LIN {X 0,Y 573.271,Z 400.076,A -85,B 0,C 180,E1 -2125.671,E2 -2125.671} C_VEL
LIN {X 0,Y 573.245,Z 400.079,A -85,B 0,C 180,E1 -2128.184,E2 -2128.184} C_VEL
LIN {X 0,Y 573.268,Z 400.071,A -85,B 0,C 180,E1 -2130.634,E2 -2130.634} C_VEL
LIN {X 0,Y 573.241,Z 400.078,A -85,B 0,C 180,E1 -2133.508,E2 -2133.508} C_VEL
LIN {X 0,Y 573.231,Z 400.08,A -85,B 0,C 180,E1 -2136.134,E2 -2136.134} C_VEL
LIN {X 0,Y 573.255,Z 400.074,A -85,B 0,C 180,E1 -2139.174,E2 -2139.174} C_VEL
LIN {X 0,Y 573.225,Z 400.08,A -85,B 0,C 180,E1 -2141.411,E2 -2141.411} C_VEL
LIN {X 0,Y 573.248,Z 400.081,A -85,B 0,C 180,E1 -2143.621,E2 -2143.621} C_VEL
LIN {X 0,Y 573.277,Z 400.078,A -85,B 0,C 180,E1 -2145.807,E2 -2145.807} C_VEL
LIN {X 0,Y 573.27,Z 400.072,A -85,B 0,C 180,E1 -2148.744,E2 -2148.744} C_VEL
LIN {X 0,Y 573.289,Z 400.17,A -85,B 0,C 180,E1 -2149.099,E2 -2149.099} C_VEL
LIN {X 0,Y 573.723,Z 402.646,A -85,B 0,C 180,E1 -2149.194,E2 -2149.194} C_VEL
LIN {X 0,Y 573.631,Z 415.712,A -85,B 0,C 180,E1 -2149.767,E2 -2149.767} C_VEL
LIN {X 0,Y 573.485,Z 426.532,A -85,B 0,C 180,E1 -2150.388,E2 -2150.388} C_VEL
LIN {X 0,Y 573.341,Z 436.494,A -85,B 0,C 180,E1 -2151.097,E2 -2151.097} C_VEL
LIN {X 0,Y 573.294,Z 445.705,A -85,B 0,C 180,E1 -2151.895,E2 -2151.895} C_VEL
LIN {X 0,Y 573.193,Z 454.155,A -85,B 0,C 180,E1 -2152.78,E2 -2152.78} C_VEL
LIN {X 0,Y 573.148,Z 462.359,A -85,B 0,C 180,E1 -2153.841,E2 -2153.841} C_VEL
LIN {X 0,Y 573.024,Z 467.955,A -85,B 0,C 180,E1 -2154.722,E2 -2154.722} C_VEL
LIN {X 0,Y 573.036,Z 473.419,A -85,B 0,C 180,E1 -2155.78,E2 -2155.78} C_VEL
LIN {X 0,Y 573.011,Z 477.698,A -85,B 0,C 180,E1 -2156.836,E2 -2156.836} C_VEL
LIN {X 0,Y 572.952,Z 480.925,A -85,B 0,C 180,E1 -2157.891,E2 -2157.891} C_VEL
LIN {X 0,Y 572.949,Z 482.571,A -85,B 0,C 180,E1 -2158.594,E2 -2158.594} C_VEL
LIN {X 0,Y 572.941,Z 483.756,A -85,B 0,C 180,E1 -2159.297,E2 -2159.297} C_VEL
LIN {X 0,Y 572.94,Z 484.933,A -85,B 0,C 180,E1 -2160.703,E2 -2160.703} C_VEL
LIN {X 0,Y 572.946,Z 484.929,A -85,B 0,C 180,E1 -2161.406,E2 -2161.406} C_VEL
LIN {X 0,Y 572.955,Z 483.726,A -85,B 0,C 180,E1 -2162.812,E2 -2162.812} C_VEL
LIN {X 0,Y 573.009,Z 482.529,A -85,B 0,C 180,E1 -2163.516,E2 -2163.516} C_VEL
LIN {X 0,Y 573.005,Z 479.934,A -85,B 0,C 180,E1 -2164.573,E2 -2164.573} C_VEL
LIN {X 0,Y 573.051,Z 476.328,A -85,B 0,C 180,E1 -2165.63,E2 -2165.63} C_VEL
LIN {X 0,Y 573.059,Z 471.604,A -85,B 0,C 180,E1 -2166.691,E2 -2166.691} C_VEL
LIN {X 0,Y 573.087,Z 465.621,A -85,B 0,C 180,E1 -2167.753,E2 -2167.753} C_VEL
LIN {X 0,Y 573.158,Z 458.145,A -85,B 0,C 180,E1 -2168.817,E2 -2168.817} C_VEL
LIN {X 0,Y 573.217,Z 450.542,A -85,B 0,C 180,E1 -2169.705,E2 -2169.705} C_VEL
LIN {X 0,Y 573.342,Z 441.353,A -85,B 0,C 180,E1 -2170.595,E2 -2170.595} C_VEL
LIN {X 0,Y 573.451,Z 430.069,A -85,B 0,C 180,E1 -2171.469,E2 -2171.469} C_VEL
LIN {X 0,Y 573.555,Z 419.634,A -85,B 0,C 180,E1 -2172.113,E2 -2172.113} C_VEL
LIN {X 0,Y 573.669,Z 407.697,A -85,B 0,C 180,E1 -2172.694,E2 -2172.694} C_VEL
LIN {X 0,Y 573.7,Z 402.018,A -85,B 0,C 180,E1 -2172.919,E2 -2172.919} C_VEL
LIN {X 0,Y 573.284,Z 400.077,A -85,B 0,C 180,E1 -2172.996,E2 -2172.996} C_VEL
LIN {X 0,Y 573.244,Z 400.08,A -85,B 0,C 180,E1 -2175.648,E2 -2175.648} C_VEL
LIN {X 0,Y 573.243,Z 400.081,A -85,B 0,C 180,E1 -2177.849,E2 -2177.849} C_VEL
LIN {X 0,Y 573.256,Z 400.082,A -85,B 0,C 180,E1 -2180.076,E2 -2180.076} C_VEL
LIN {X 0,Y 573.239,Z 400.084,A -85,B 0,C 180,E1 -2183.099,E2 -2183.099} C_VEL
LIN {X 0,Y 573.26,Z 400.078,A -85,B 0,C 180,E1 -2185.41,E2 -2185.41} C_VEL
LIN {X 0,Y 573.257,Z 400.077,A -85,B 0,C 180,E1 -2188.029,E2 -2188.029} C_VEL
LIN {X 0,Y 573.251,Z 400.081,A -85,B 0,C 180,E1 -2190.176,E2 -2190.176} C_VEL
LIN {X 0,Y 573.258,Z 400.081,A -85,B 0,C 180,E1 -2192.645,E2 -2192.645} C_VEL
LIN {X 0,Y 573.211,Z 400.084,A -85,B 0,C 180,E1 -2195.188,E2 -2195.188} C_VEL
LIN {X 0,Y 573.238,Z 400.08,A -85,B 0,C 180,E1 -2197.807,E2 -2197.807} C_VEL
LIN {X 0,Y 573.248,Z 400.079,A -85,B 0,C 180,E1 -2200.525,E2 -2200.525} C_VEL
LIN {X 0,Y 573.252,Z 400.078,A -85,B 0,C 180,E1 -2203.358,E2 -2203.358} C_VEL
LIN {X 0,Y 573.243,Z 400.08,A -85,B 0,C 180,E1 -2206.331,E2 -2206.331} C_VEL
LIN {X 0,Y 573.274,Z 400.079,A -85,B 0,C 180,E1 -2209.472,E2 -2209.472} C_VEL
LIN {X 0,Y 573.24,Z 400.084,A -85,B 0,C 180,E1 -2212.192,E2 -2212.192} C_VEL
LIN {X 0,Y 573.309,Z 400.2,A -85,B 0,C 180,E1 -2213.383,E2 -2213.383} C_VEL
LIN {X 0,Y 573.995,Z 405.053,A -85,B 0,C 180,E1 -2214.437,E2 -2214.437} C_VEL
LIN {X 0,Y 573.917,Z 418.715,A -85,B 0,C 180,E1 -2217.189,E2 -2217.189} C_VEL
LIN {X 0,Y 573.925,Z 434.068,A -85,B 0,C 180,E1 -2220.168,E2 -2220.168} C_VEL
LIN {X 0,Y 573.92,Z 449.451,A -85,B 0,C 180,E1 -2223.058,E2 -2223.058} C_VEL
LIN {X 0,Y 573.821,Z 461.449,A -85,B 0,C 180,E1 -2225.391,E2 -2225.391} C_VEL
LIN {X 0,Y 573.637,Z 475.144,A -85,B 0,C 180,E1 -2228.057,E2 -2228.057} C_VEL
LIN {X 0,Y 573.502,Z 488.839,A -85,B 0,C 180,E1 -2230.678,E2 -2230.678} C_VEL
LIN {X 0,Y 573.363,Z 502.686,A -85,B 0,C 180,E1 -2233.287,E2 -2233.287} C_VEL
LIN {X 0,Y 573.252,Z 518.186,A -85,B 0,C 180,E1 -2236.168,E2 -2236.168} C_VEL
LIN {X 0,Y 573.191,Z 525.155,A -85,B 0,C 180,E1 -2237.452,E2 -2237.452} C_VEL
LIN {X 0,Y 573.863,Z 530.936,A -85,B 0,C 180,E1 -2237.557,E2 -2237.557} C_VEL
LIN {X 0,Y 573.81,Z 544.212,A -85,B 0,C 180,E1 -2237.87,E2 -2237.87} C_VEL
LIN {X 0,Y 573.714,Z 556.368,A -85,B 0,C 180,E1 -2238.294,E2 -2238.294} C_VEL
LIN {X 0,Y 573.586,Z 568.658,A -85,B 0,C 180,E1 -2238.875,E2 -2238.875} C_VEL
LIN {X 0,Y 573.434,Z 580.2,A -85,B 0,C 180,E1 -2239.585,E2 -2239.585} C_VEL
LIN {X 0,Y 573.334,Z 590.597,A -85,B 0,C 180,E1 -2240.385,E2 -2240.385} C_VEL
LIN {X 0,Y 573.241,Z 599.11,A -85,B 0,C 180,E1 -2241.184,E2 -2241.184} C_VEL
LIN {X 0,Y 573.161,Z 606.959,A -85,B 0,C 180,E1 -2242.071,E2 -2242.071} C_VEL
LIN {X 0,Y 573.073,Z 614.953,A -85,B 0,C 180,E1 -2243.185,E2 -2243.185} C_VEL
LIN {X 0,Y 573.07,Z 621.679,A -85,B 0,C 180,E1 -2244.369,E2 -2244.369} C_VEL
LIN {X 0,Y 573.029,Z 626.371,A -85,B 0,C 180,E1 -2245.427,E2 -2245.427} C_VEL
LIN {X 0,Y 573.022,Z 629.956,A -85,B 0,C 180,E1 -2246.484,E2 -2246.484} C_VEL
LIN {X 0,Y 572.959,Z 631.808,A -85,B 0,C 180,E1 -2247.188,E2 -2247.188} C_VEL
LIN {X 0,Y 572.938,Z 633.199,A -85,B 0,C 180,E1 -2247.891,E2 -2247.891} C_VEL
LIN {X 0,Y 572.941,Z 634.785,A -85,B 0,C 180,E1 -2249.297,E2 -2249.297} C_VEL
LIN {X 0,Y 572.938,Z 635,A -85,B 0,C 180,E1 -2250,E2 -2250} C_VEL
LIN {X 0,Y 572.946,Z 634.186,A -85,B 0,C 180,E1 -2251.406,E2 -2251.406} C_VEL
LIN {X 0,Y 572.938,Z 633.2,A -85,B 0,C 180,E1 -2252.109,E2 -2252.109} C_VEL
LIN {X 0,Y 572.959,Z 631.81,A -85,B 0,C 180,E1 -2252.812,E2 -2252.812} C_VEL
LIN {X 0,Y 573.014,Z 628.896,A -85,B 0,C 180,E1 -2253.868,E2 -2253.868} C_VEL
LIN {X 0,Y 572.963,Z 624.95,A -85,B 0,C 180,E1 -2254.925,E2 -2254.925} C_VEL
LIN {X 0,Y 573.064,Z 618.878,A -85,B 0,C 180,E1 -2256.16,E2 -2256.16} C_VEL
LIN {X 0,Y 573.119,Z 612.238,A -85,B 0,C 180,E1 -2257.221,E2 -2257.221} C_VEL
LIN {X 0,Y 573.201,Z 603.991,A -85,B 0,C 180,E1 -2258.283,E2 -2258.283} C_VEL
LIN {X 0,Y 573.287,Z 595.539,A -85,B 0,C 180,E1 -2259.17,E2 -2259.17} C_VEL
LIN {X 0,Y 573.42,Z 585.098,A -85,B 0,C 180,E1 -2260.058,E2 -2260.058} C_VEL
LIN {X 0,Y 573.555,Z 573.44,A -85,B 0,C 180,E1 -2260.852,E2 -2260.852} C_VEL
LIN {X 0,Y 573.65,Z 562.318,A -85,B 0,C 180,E1 -2261.446,E2 -2261.446} C_VEL
LIN {X 0,Y 573.731,Z 549.177,A -85,B 0,C 180,E1 -2261.974,E2 -2261.974} C_VEL
LIN {X 0,Y 573.854,Z 536.524,A -85,B 0,C 180,E1 -2262.331,E2 -2262.331} C_VEL
LIN {X 0,Y 573.611,Z 527.738,A -85,B 0,C 180,E1 -2262.499,E2 -2262.499} C_VEL
LIN {X 0,Y 573.194,Z 525.035,A -85,B 0,C 180,E1 -2262.57,E2 -2262.57} C_VEL
LIN {X 0,Y 573.316,Z 510.362,A -85,B 0,C 180,E1 -2265.281,E2 -2265.281} C_VEL
LIN {X 0,Y 573.46,Z 494.71,A -85,B 0,C 180,E1 -2268.211,E2 -2268.211} C_VEL
LIN {X 0,Y 573.597,Z 479.542,A -85,B 0,C 180,E1 -2271.096,E2 -2271.096} C_VEL
LIN {X 0,Y 573.775,Z 465.364,A -85,B 0,C 180,E1 -2273.841,E2 -2273.841} C_VEL
LIN {X 0,Y 573.939,Z 451.13,A -85,B 0,C 180,E1 -2276.632,E2 -2276.632} C_VEL
LIN {X 0,Y 573.94,Z 435.25,A -85,B 0,C 180,E1 -2279.61,E2 -2279.61} C_VEL
LIN {X 0,Y 573.92,Z 421.222,A -85,B 0,C 180,E1 -2282.333,E2 -2282.333} C_VEL
LIN {X 0,Y 574.045,Z 405.153,A -85,B 0,C 180,E1 -2285.559,E2 -2285.559} C_VEL
LIN {X 0,Y 573.294,Z 400.077,A -85,B 0,C 180,E1 -2286.7,E2 -2286.7} C_VEL
LIN {X 0,Y 573.251,Z 400.081,A -85,B 0,C 180,E1 -2289.607,E2 -2289.607} C_VEL
LIN {X 0,Y 573.242,Z 400.084,A -85,B 0,C 180,E1 -2292.641,E2 -2292.641} C_VEL
LIN {X 0,Y 573.242,Z 400.084,A -85,B 0,C 180,E1 -2295.667,E2 -2295.667} C_VEL
LIN {X 0,Y 573.247,Z 400.081,A -85,B 0,C 180,E1 -2298.544,E2 -2298.544} C_VEL
LIN {X 0,Y 573.252,Z 400.082,A -85,B 0,C 180,E1 -2301.299,E2 -2301.299} C_VEL
LIN {X 0,Y 573.244,Z 400.081,A -85,B 0,C 180,E1 -2304.014,E2 -2304.014} C_VEL
LIN {X 0,Y 573.271,Z 400.08,A -85,B 0,C 180,E1 -2306.518,E2 -2306.518} C_VEL
LIN {X 0,Y 573.231,Z 400.082,A -85,B 0,C 180,E1 -2309.118,E2 -2309.118} C_VEL
LIN {X 0,Y 573.266,Z 400.08,A -85,B 0,C 180,E1 -2311.969,E2 -2311.969} C_VEL
LIN {X 0,Y 573.26,Z 400.079,A -85,B 0,C 180,E1 -2314.59,E2 -2314.59} C_VEL
LIN {X 0,Y 573.24,Z 400.083,A -85,B 0,C 180,E1 -2317.662,E2 -2317.662} C_VEL
LIN {X 0,Y 573.281,Z 400.078,A -85,B 0,C 180,E1 -2320.728,E2 -2320.728} C_VEL
LIN {X 0,Y 573.257,Z 400.079,A -85,B 0,C 180,E1 -2323.622,E2 -2323.622} C_VEL
LIN {X 0,Y 573.277,Z 400.077,A -85,B 0,C 180,E1 -2325.807,E2 -2325.807} C_VEL
LIN {X 0,Y 573.265,Z 400.078,A -85,B 0,C 180,E1 -2328.745,E2 -2328.745} C_VEL
LIN {X 0,Y 573.257,Z 400.081,A -85,B 0,C 180,E1 -2331.54,E2 -2331.54} C_VEL
LIN {X 0,Y 573.248,Z 400.082,A -85,B 0,C 180,E1 -2333.665,E2 -2333.665} C_VEL
LIN {X 0,Y 573.234,Z 400.084,A -85,B 0,C 180,E1 -2335.782,E2 -2335.782} C_VEL
LIN {X 0,Y 573.317,Z 400.073,A -85,B 0,C 180,E1 -2337.893,E2 -2337.893} C_VEL
LIN {X 0,Y 573.337,Z 400.069,A -85,B 0,C 180,E1 -2340.702,E2 -2340.702} C_VEL
LIN {X 0,Y 573.235,Z 400.085,A -85,B 0,C 180,E1 -2343.515,E2 -2343.515} C_VEL
LIN {X 0,Y 573.291,Z 400.078,A -85,B 0,C 180,E1 -2345.628,E2 -2345.628} C_VEL
LIN {X 0,Y 573.294,Z 400.075,A -85,B 0,C 180,E1 -2348.46,E2 -2348.46} C_VEL
LIN {X 0,Y 573.275,Z 400.078,A -85,B 0,C 180,E1 -2351.312,E2 -2351.312} C_VEL
LIN {X 0,Y 573.277,Z 400.079,A -85,B 0,C 180,E1 -2354.193,E2 -2354.193} C_VEL
LIN {X 0,Y 573.261,Z 400.078,A -85,B 0,C 180,E1 -2357.112,E2 -2357.112} C_VEL
LIN {X 0,Y 573.259,Z 400.079,A -85,B 0,C 180,E1 -2360.077,E2 -2360.077} C_VEL
LIN {X 0,Y 573.242,Z 400.081,A -85,B 0,C 180,E1 -2362.338,E2 -2362.338} C_VEL
LIN {X 0,Y 573.254,Z 400.078,A -85,B 0,C 180,E1 -2364.393,E2 -2364.393} C_VEL
LIN {X 0,Y 572.627,Z 400.159,A -85,B 0,C 180,E1 -2364.98,E2 -2364.98} C_VEL
LIN {X 0,Y 569.784,Z 400.516,A -85,B 0,C 180,E1 -2365.931,E2 -2365.931} C_VEL
LIN {X 0,Y 567.351,Z 400.819,A -85,B 0,C 180,E1 -2366.697,E2 -2366.697} C_VEL
LIN {X 0,Y 566.296,Z 400.949,A -85,B 0,C 180,E1 -2367.288,E2 -2367.288} C_VEL
LIN {X 0,Y 566.206,Z 400.959,A -85,B 0,C 180,E1 -2367.488,E2 -2367.488} C_VEL
LIN {X 0,Y 566.204,Z 400.959,A -85,B 0,C 180,E1 -2369.769,E2 -2369.769} C_VEL
LIN {X 0,Y 566.209,Z 400.958,A -85,B 0,C 180,E1 -2372.431,E2 -2372.431} C_VEL
LIN {X 0,Y 566.206,Z 400.959,A -85,B 0,C 180,E1 -2374.993,E2 -2374.993} C_VEL
LIN {X 0,Y 566.2,Z 400.958,A -85,B 0,C 180,E1 -2377.461,E2 -2377.461} C_VEL
LIN {X 0,Y 566.21,Z 400.959,A -85,B 0,C 180,E1 -2380.199,E2 -2380.199} C_VEL
LIN {X 0,Y 566.209,Z 400.957,A -85,B 0,C 180,E1 -2383.054,E2 -2383.054} C_VEL
LIN {X 0,Y 566.206,Z 400.958,A -85,B 0,C 180,E1 -2386.048,E2 -2386.048} C_VEL
LIN {X 0,Y 566.215,Z 400.958,A -85,B 0,C 180,E1 -2388.864,E2 -2388.864} C_VEL
LIN {X 0,Y 566.193,Z 400.959,A -85,B 0,C 180,E1 -2391.637,E2 -2391.637} C_VEL
LIN {X 0,Y 566.204,Z 400.96,A -85,B 0,C 180,E1 -2394.311,E2 -2394.311} C_VEL
LIN {X 0,Y 566.234,Z 400.954,A -85,B 0,C 180,E1 -2396.899,E2 -2396.899} C_VEL
LIN {X 0,Y 566.199,Z 400.959,A -85,B 0,C 180,E1 -2399.408,E2 -2399.408} C_VEL
LIN {X 0,Y 566.216,Z 400.959,A -85,B 0,C 180,E1 -2401.858,E2 -2401.858} C_VEL
LIN {X 0,Y 566.217,Z 400.957,A -85,B 0,C 180,E1 -2404.251,E2 -2404.251} C_VEL
LIN {X 0,Y 566.178,Z 400.96,A -85,B 0,C 180,E1 -2406.718,E2 -2406.718} C_VEL
LIN {X 0,Y 566.219,Z 400.958,A -85,B 0,C 180,E1 -2409.663,E2 -2409.663} C_VEL
LIN {X 0,Y 566.208,Z 400.959,A -85,B 0,C 180,E1 -2412.669,E2 -2412.669} C_VEL
LIN {X 0,Y 566.239,Z 400.954,A -85,B 0,C 180,E1 -2415.627,E2 -2415.627} C_VEL
LIN {X 0,Y 566.24,Z 400.953,A -85,B 0,C 180,E1 -2418.675,E2 -2418.675} C_VEL
LIN {X 0,Y 566.232,Z 400.955,A -85,B 0,C 180,E1 -2420.962,E2 -2420.962} C_VEL
LIN {X 0,Y 566.753,Z 404.787,A -85,B 0,C 180,E1 -2421.128,E2 -2421.128} C_VEL
LIN {X 0,Y 566.621,Z 417.32,A -85,B 0,C 180,E1 -2421.71,E2 -2421.71} C_VEL
LIN {X 0,Y 566.484,Z 427.742,A -85,B 0,C 180,E1 -2422.336,E2 -2422.336} C_VEL
LIN {X 0,Y 566.34,Z 436.703,A -85,B 0,C 180,E1 -2422.99,E2 -2422.99} C_VEL
LIN {X 0,Y 566.196,Z 445.6,A -85,B 0,C 180,E1 -2423.765,E2 -2423.765} C_VEL
LIN {X 0,Y 566.157,Z 455.476,A -85,B 0,C 180,E1 -2424.837,E2 -2424.837} C_VEL
LIN {X 0,Y 566.084,Z 463.43,A -85,B 0,C 180,E1 -2425.906,E2 -2425.906} C_VEL
LIN {X 0,Y 566.013,Z 468.831,A -85,B 0,C 180,E1 -2426.797,E2 -2426.797} C_VEL
LIN {X 0,Y 565.885,Z 474.122,A -85,B 0,C 180,E1 -2427.865,E2 -2427.865} C_VEL
LIN {X 0,Y 565.912,Z 478.247,A -85,B 0,C 180,E1 -2428.933,E2 -2428.933} C_VEL
LIN {X 0,Y 565.844,Z 481.333,A -85,B 0,C 180,E1 -2430,E2 -2430} C_VEL
LIN {X 0,Y 565.841,Z 482.847,A -85,B 0,C 180,E1 -2430.712,E2 -2430.712} C_VEL
LIN {X 0,Y 565.839,Z 484.657,A -85,B 0,C 180,E1 -2432.136,E2 -2432.136} C_VEL
LIN {X 0,Y 565.911,Z 484.894,A -85,B 0,C 180,E1 -2433.56,E2 -2433.56} C_VEL
LIN {X 0,Y 565.912,Z 484.393,A -85,B 0,C 180,E1 -2434.273,E2 -2434.273} C_VEL
LIN {X 0,Y 565.851,Z 483.503,A -85,B 0,C 180,E1 -2434.988,E2 -2434.988} C_VEL
LIN {X 0,Y 565.899,Z 480.492,A -85,B 0,C 180,E1 -2436.418,E2 -2436.418} C_VEL
LIN {X 0,Y 565.922,Z 477.065,A -85,B 0,C 180,E1 -2437.493,E2 -2437.493} C_VEL
LIN {X 0,Y 565.954,Z 472.52,A -85,B 0,C 180,E1 -2438.57,E2 -2438.57} C_VEL
LIN {X 0,Y 566.005,Z 466.736,A -85,B 0,C 180,E1 -2439.65,E2 -2439.65} C_VEL
LIN {X 0,Y 566.064,Z 459.561,A -85,B 0,C 180,E1 -2440.733,E2 -2440.733} C_VEL
LIN {X 0,Y 566.191,Z 450.536,A -85,B 0,C 180,E1 -2441.819,E2 -2441.819} C_VEL
LIN {X 0,Y 566.295,Z 441.228,A -85,B 0,C 180,E1 -2442.726,E2 -2442.726} C_VEL
LIN {X 0,Y 566.42,Z 430.825,A -85,B 0,C 180,E1 -2443.544,E2 -2443.544} C_VEL
LIN {X 0,Y 566.56,Z 420.83,A -85,B 0,C 180,E1 -2444.182,E2 -2444.182} C_VEL
LIN {X 0,Y 566.719,Z 409.031,A -85,B 0,C 180,E1 -2444.784,E2 -2444.784} C_VEL
LIN {X 0,Y 566.786,Z 403.376,A -85,B 0,C 180,E1 -2445.016,E2 -2445.016} C_VEL
LIN {X 0,Y 566.244,Z 400.951,A -85,B 0,C 180,E1 -2445.131,E2 -2445.131} C_VEL
LIN {X 0,Y 566.2,Z 400.957,A -85,B 0,C 180,E1 -2448.078,E2 -2448.078} C_VEL
LIN {X 0,Y 566.213,Z 400.959,A -85,B 0,C 180,E1 -2450.337,E2 -2450.337} C_VEL
LIN {X 0,Y 566.175,Z 400.954,A -85,B 0,C 180,E1 -2453.281,E2 -2453.281} C_VEL
LIN {X 0,Y 566.219,Z 400.951,A -85,B 0,C 180,E1 -2455.749,E2 -2455.749} C_VEL
LIN {X 0,Y 566.208,Z 400.959,A -85,B 0,C 180,E1 -2458.202,E2 -2458.202} C_VEL
LIN {X 0,Y 566.196,Z 400.952,A -85,B 0,C 180,E1 -2461.076,E2 -2461.076} C_VEL
LIN {X 0,Y 566.218,Z 400.951,A -85,B 0,C 180,E1 -2463.734,E2 -2463.734} C_VEL
LIN {X 0,Y 566.213,Z 400.953,A -85,B 0,C 180,E1 -2466.569,E2 -2466.569} C_VEL
LIN {X 0,Y 566.221,Z 400.951,A -85,B 0,C 180,E1 -2469.686,E2 -2469.686} C_VEL
LIN {X 0,Y 566.206,Z 400.95,A -85,B 0,C 180,E1 -2472.917,E2 -2472.917} C_VEL
LIN {X 0,Y 566.208,Z 400.96,A -85,B 0,C 180,E1 -2476.048,E2 -2476.048} C_VEL
LIN {X 0,Y 566.187,Z 400.953,A -85,B 0,C 180,E1 -2478.861,E2 -2478.861} C_VEL
LIN {X 0,Y 566.19,Z 400.956,A -85,B 0,C 180,E1 -2481.637,E2 -2481.637} C_VEL
LIN {X 0,Y 566.167,Z 400.959,A -85,B 0,C 180,E1 -2484.308,E2 -2484.308} C_VEL
LIN {X 0,Y 566.225,Z 400.948,A -85,B 0,C 180,E1 -2486.898,E2 -2486.898} C_VEL
LIN {X 0,Y 566.185,Z 400.955,A -85,B 0,C 180,E1 -2489.407,E2 -2489.407} C_VEL
LIN {X 0,Y 566.217,Z 400.959,A -85,B 0,C 180,E1 -2491.857,E2 -2491.857} C_VEL
LIN {X 0,Y 566.218,Z 400.952,A -85,B 0,C 180,E1 -2494.251,E2 -2494.251} C_VEL
LIN {X 0,Y 566.173,Z 400.954,A -85,B 0,C 180,E1 -2496.719,E2 -2496.719} C_VEL
LIN {X 0,Y 566.212,Z 400.958,A -85,B 0,C 180,E1 -2499.663,E2 -2499.663} C_VEL
LIN {X 0,Y 566.204,Z 400.95,A -85,B 0,C 180,E1 -2502.668,E2 -2502.668} C_VEL
LIN {X 0,Y 566.239,Z 400.955,A -85,B 0,C 180,E1 -2505.627,E2 -2505.627} C_VEL
LIN {X 0,Y 566.242,Z 400.948,A -85,B 0,C 180,E1 -2508.674,E2 -2508.674} C_VEL
LIN {X 0,Y 566.239,Z 401.02,A -85,B 0,C 180,E1 -2508.978,E2 -2508.978} C_VEL
LIN {X 0,Y 566.766,Z 403.757,A -85,B 0,C 180,E1 -2509.087,E2 -2509.087} C_VEL
LIN {X 0,Y 566.661,Z 415.97,A -85,B 0,C 180,E1 -2509.64,E2 -2509.64} C_VEL
LIN {X 0,Y 566.506,Z 426.717,A -85,B 0,C 180,E1 -2510.268,E2 -2510.268} C_VEL
LIN {X 0,Y 566.338,Z 436.65,A -85,B 0,C 180,E1 -2510.986,E2 -2510.986} C_VEL
LIN {X 0,Y 566.262,Z 445.838,A -85,B 0,C 180,E1 -2511.794,E2 -2511.794} C_VEL
LIN {X 0,Y 566.119,Z 455.757,A -85,B 0,C 180,E1 -2512.869,E2 -2512.869} C_VEL
LIN {X 0,Y 566.084,Z 463.615,A -85,B 0,C 180,E1 -2513.942,E2 -2513.942} C_VEL
LIN {X 0,Y 565.915,Z 469.96,A -85,B 0,C 180,E1 -2515.013,E2 -2515.013} C_VEL
LIN {X 0,Y 565.947,Z 475.023,A -85,B 0,C 180,E1 -2516.084,E2 -2516.084} C_VEL
LIN {X 0,Y 565.914,Z 480.041,A -85,B 0,C 180,E1 -2517.509,E2 -2517.509} C_VEL
LIN {X 0,Y 565.849,Z 482.599,A -85,B 0,C 180,E1 -2518.576,E2 -2518.576} C_VEL
LIN {X 0,Y 565.841,Z 483.775,A -85,B 0,C 180,E1 -2519.288,E2 -2519.288} C_VEL
LIN {X 0,Y 565.84,Z 484.936,A -85,B 0,C 180,E1 -2520.712,E2 -2520.712} C_VEL
LIN {X 0,Y 565.846,Z 484.927,A -85,B 0,C 180,E1 -2521.423,E2 -2521.423} C_VEL
LIN {X 0,Y 565.874,Z 483.704,A -85,B 0,C 180,E1 -2522.847,E2 -2522.847} C_VEL
LIN {X 0,Y 565.915,Z 482.505,A -85,B 0,C 180,E1 -2523.56,E2 -2523.56} C_VEL
LIN {X 0,Y 565.896,Z 479.897,A -85,B 0,C 180,E1 -2524.63,E2 -2524.63} C_VEL
LIN {X 0,Y 565.978,Z 476.278,A -85,B 0,C 180,E1 -2525.701,E2 -2525.701} C_VEL
LIN {X 0,Y 565.973,Z 470.712,A -85,B 0,C 180,E1 -2526.936,E2 -2526.936} C_VEL
LIN {X 0,Y 566.022,Z 464.381,A -85,B 0,C 180,E1 -2528.03,E2 -2528.03} C_VEL
LIN {X 0,Y 566.108,Z 458.035,A -85,B 0,C 180,E1 -2528.927,E2 -2528.927} C_VEL
LIN {X 0,Y 566.189,Z 450.414,A -85,B 0,C 180,E1 -2529.827,E2 -2529.827} C_VEL
LIN {X 0,Y 566.324,Z 441.203,A -85,B 0,C 180,E1 -2530.728,E2 -2530.728} C_VEL
LIN {X 0,Y 566.46,Z 429.586,A -85,B 0,C 180,E1 -2531.631,E2 -2531.631} C_VEL
LIN {X 0,Y 566.571,Z 419.374,A -85,B 0,C 180,E1 -2532.265,E2 -2532.265} C_VEL
LIN {X 0,Y 566.703,Z 408.396,A -85,B 0,C 180,E1 -2532.808,E2 -2532.808} C_VEL
LIN {X 0,Y 566.671,Z 402.914,A -85,B 0,C 180,E1 -2533.036,E2 -2533.036} C_VEL
LIN {X 0,Y 566.221,Z 400.958,A -85,B 0,C 180,E1 -2533.138,E2 -2533.138} C_VEL
LIN {X 0,Y 566.21,Z 400.958,A -85,B 0,C 180,E1 -2535.847,E2 -2535.847} C_VEL
LIN {X 0,Y 566.197,Z 400.958,A -85,B 0,C 180,E1 -2538.078,E2 -2538.078} C_VEL
LIN {X 0,Y 566.218,Z 400.959,A -85,B 0,C 180,E1 -2540.337,E2 -2540.337} C_VEL
LIN {X 0,Y 566.173,Z 400.962,A -85,B 0,C 180,E1 -2543.281,E2 -2543.281} C_VEL
LIN {X 0,Y 566.22,Z 400.958,A -85,B 0,C 180,E1 -2545.749,E2 -2545.749} C_VEL
LIN {X 0,Y 566.207,Z 400.956,A -85,B 0,C 180,E1 -2548.202,E2 -2548.202} C_VEL
LIN {X 0,Y 566.195,Z 400.959,A -85,B 0,C 180,E1 -2551.076,E2 -2551.076} C_VEL
LIN {X 0,Y 566.216,Z 400.955,A -85,B 0,C 180,E1 -2553.734,E2 -2553.734} C_VEL
LIN {X 0,Y 566.204,Z 400.957,A -85,B 0,C 180,E1 -2556.57,E2 -2556.57} C_VEL
LIN {X 0,Y 566.219,Z 400.958,A -85,B 0,C 180,E1 -2559.686,E2 -2559.686} C_VEL
LIN {X 0,Y 566.21,Z 400.956,A -85,B 0,C 180,E1 -2562.918,E2 -2562.918} C_VEL
LIN {X 0,Y 566.198,Z 400.956,A -85,B 0,C 180,E1 -2566.049,E2 -2566.049} C_VEL
LIN {X 0,Y 566.224,Z 400.956,A -85,B 0,C 180,E1 -2569.212,E2 -2569.212} C_VEL
LIN {X 0,Y 566.193,Z 400.959,A -85,B 0,C 180,E1 -2571.637,E2 -2571.637} C_VEL
LIN {X 0,Y 566.245,Z 401.004,A -85,B 0,C 180,E1 -2573.156,E2 -2573.156} C_VEL
LIN {X 0,Y 567.071,Z 406.484,A -85,B 0,C 180,E1 -2574.373,E2 -2574.373} C_VEL
LIN {X 0,Y 566.969,Z 419.054,A -85,B 0,C 180,E1 -2576.947,E2 -2576.947} C_VEL
LIN {X 0,Y 566.974,Z 433.91,A -85,B 0,C 180,E1 -2579.866,E2 -2579.866} C_VEL
LIN {X 0,Y 566.924,Z 448.675,A -85,B 0,C 180,E1 -2582.698,E2 -2582.698} C_VEL
LIN {X 0,Y 566.852,Z 463.406,A -85,B 0,C 180,E1 -2585.459,E2 -2585.459} C_VEL
LIN {X 0,Y 566.653,Z 477.101,A -85,B 0,C 180,E1 -2588.156,E2 -2588.156} C_VEL
LIN {X 0,Y 566.494,Z 491.063,A -85,B 0,C 180,E1 -2590.858,E2 -2590.858} C_VEL
LIN {X 0,Y 566.335,Z 504.491,A -85,B 0,C 180,E1 -2593.416,E2 -2593.416} C_VEL
LIN {X 0,Y 566.198,Z 520.142,A -85,B 0,C 180,E1 -2596.359,E2 -2596.359} C_VEL
LIN {X 0,Y 566.153,Z 525.11,A -85,B 0,C 180,E1 -2597.285,E2 -2597.285} C_VEL
LIN {X 0,Y 566.954,Z 532.077,A -85,B 0,C 180,E1 -2597.425,E2 -2597.425} C_VEL
LIN {X 0,Y 566.831,Z 545.732,A -85,B 0,C 180,E1 -2597.764,E2 -2597.764} C_VEL
LIN {X 0,Y 566.706,Z 558.519,A -85,B 0,C 180,E1 -2598.238,E2 -2598.238} C_VEL
LIN {X 0,Y 566.561,Z 570.723,A -85,B 0,C 180,E1 -2598.853,E2 -2598.853} C_VEL
LIN {X 0,Y 566.419,Z 581.479,A -85,B 0,C 180,E1 -2599.545,E2 -2599.545} C_VEL
LIN {X 0,Y 566.301,Z 591.645,A -85,B 0,C 180,E1 -2600.355,E2 -2600.355} C_VEL
LIN {X 0,Y 566.166,Z 600.785,A -85,B 0,C 180,E1 -2601.253,E2 -2601.253} C_VEL
LIN {X 0,Y 566.081,Z 609.688,A -85,B 0,C 180,E1 -2602.33,E2 -2602.33} C_VEL
LIN {X 0,Y 565.968,Z 616.955,A -85,B 0,C 180,E1 -2603.422,E2 -2603.422} C_VEL
LIN {X 0,Y 566.004,Z 621.679,A -85,B 0,C 180,E1 -2604.299,E2 -2604.299} C_VEL
LIN {X 0,Y 565.933,Z 626.371,A -85,B 0,C 180,E1 -2605.37,E2 -2605.37} C_VEL
LIN {X 0,Y 565.927,Z 629.957,A -85,B 0,C 180,E1 -2606.44,E2 -2606.44} C_VEL
LIN {X 0,Y 565.878,Z 631.808,A -85,B 0,C 180,E1 -2607.152,E2 -2607.152} C_VEL
LIN {X 0,Y 565.846,Z 634.185,A -85,B 0,C 180,E1 -2608.576,E2 -2608.576} C_VEL
LIN {X 0,Y 565.839,Z 635,A -85,B 0,C 180,E1 -2610,E2 -2610} C_VEL
LIN {X 0,Y 565.846,Z 634.186,A -85,B 0,C 180,E1 -2611.423,E2 -2611.423} C_VEL
LIN {X 0,Y 565.878,Z 631.81,A -85,B 0,C 180,E1 -2612.847,E2 -2612.847} C_VEL
LIN {X 0,Y 565.926,Z 628.896,A -85,B 0,C 180,E1 -2613.916,E2 -2613.916} C_VEL
LIN {X 0,Y 565.878,Z 624.95,A -85,B 0,C 180,E1 -2614.987,E2 -2614.987} C_VEL
LIN {X 0,Y 566.002,Z 619.867,A -85,B 0,C 180,E1 -2616.058,E2 -2616.058} C_VEL
LIN {X 0,Y 566.04,Z 613.469,A -85,B 0,C 180,E1 -2617.132,E2 -2617.132} C_VEL
LIN {X 0,Y 566.133,Z 605.479,A -85,B 0,C 180,E1 -2618.208,E2 -2618.208} C_VEL
LIN {X 0,Y 566.229,Z 597.337,A -85,B 0,C 180,E1 -2619.105,E2 -2619.105} C_VEL
LIN {X 0,Y 566.342,Z 587.402,A -85,B 0,C 180,E1 -2620.005,E2 -2620.005} C_VEL
LIN {X 0,Y 566.528,Z 576.292,A -85,B 0,C 180,E1 -2620.807,E2 -2620.807} C_VEL
LIN {X 0,Y 566.612,Z 565.179,A -85,B 0,C 180,E1 -2621.447,E2 -2621.447} C_VEL
LIN {X 0,Y 566.73,Z 552.987,A -85,B 0,C 180,E1 -2621.988,E2 -2621.988} C_VEL
LIN {X 0,Y 566.887,Z 540.181,A -85,B 0,C 180,E1 -2622.394,E2 -2622.394} C_VEL
LIN {X 0,Y 566.761,Z 528.952,A -85,B 0,C 180,E1 -2622.634,E2 -2622.634} C_VEL
LIN {X 0,Y 566.155,Z 525.035,A -85,B 0,C 180,E1 -2622.729,E2 -2622.729} C_VEL
LIN {X 0,Y 566.283,Z 510.362,A -85,B 0,C 180,E1 -2625.476,E2 -2625.476} C_VEL
LIN {X 0,Y 566.459,Z 494.71,A -85,B 0,C 180,E1 -2628.444,E2 -2628.444} C_VEL
LIN {X 0,Y 566.61,Z 479.879,A -85,B 0,C 180,E1 -2631.303,E2 -2631.303} C_VEL
LIN {X 0,Y 566.812,Z 467.322,A -85,B 0,C 180,E1 -2633.764,E2 -2633.764} C_VEL
LIN {X 0,Y 566.898,Z 457.181,A -85,B 0,C 180,E1 -2635.716,E2 -2635.716} C_VEL
LIN {X 0,Y 566.935,Z 441.919,A -85,B 0,C 180,E1 -2638.584,E2 -2638.584} C_VEL
LIN {X 0,Y 566.972,Z 427.582,A -85,B 0,C 180,E1 -2641.374,E2 -2641.374} C_VEL
LIN {X 0,Y 567.049,Z 411.805,A -85,B 0,C 180,E1 -2644.543,E2 -2644.543} C_VEL
LIN {X 0,Y 567.006,Z 405.049,A -85,B 0,C 180,E1 -2645.949,E2 -2645.949} C_VEL
LIN {X 0,Y 566.226,Z 400.958,A -85,B 0,C 180,E1 -2646.901,E2 -2646.901} C_VEL
LIN {X 0,Y 566.216,Z 400.957,A -85,B 0,C 180,E1 -2649.686,E2 -2649.686} C_VEL
LIN {X 0,Y 566.193,Z 400.959,A -85,B 0,C 180,E1 -2652.089,E2 -2652.089} C_VEL
LIN {X 0,Y 566.175,Z 400.963,A -85,B 0,C 180,E1 -2655.036,E2 -2655.036} C_VEL
LIN {X 0,Y 566.217,Z 400.958,A -85,B 0,C 180,E1 -2657.913,E2 -2657.913} C_VEL
LIN {X 0,Y 566.225,Z 400.955,A -85,B 0,C 180,E1 -2660.727,E2 -2660.727} C_VEL
LIN {X 0,Y 566.207,Z 400.958,A -85,B 0,C 180,E1 -2663.785,E2 -2663.785} C_VEL
LIN {X 0,Y 566.213,Z 400.957,A -85,B 0,C 180,E1 -2666.266,E2 -2666.266} C_VEL
LIN {X 0,Y 566.193,Z 400.96,A -85,B 0,C 180,E1 -2668.923,E2 -2668.923} C_VEL
LIN {X 0,Y 566.231,Z 400.955,A -85,B 0,C 180,E1 -2671.858,E2 -2671.858} C_VEL
LIN {X 0,Y 566.229,Z 400.957,A -85,B 0,C 180,E1 -2674.252,E2 -2674.252} C_VEL
LIN {X 0,Y 566.193,Z 400.959,A -85,B 0,C 180,E1 -2676.714,E2 -2676.714} C_VEL
LIN {X 0,Y 566.215,Z 400.959,A -85,B 0,C 180,E1 -2679.663,E2 -2679.663} C_VEL
LIN {X 0,Y 566.202,Z 400.959,A -85,B 0,C 180,E1 -2682.668,E2 -2682.668} C_VEL
LIN {X 0,Y 566.237,Z 400.954,A -85,B 0,C 180,E1 -2685.627,E2 -2685.627} C_VEL
LIN {X 0,Y 566.237,Z 400.954,A -85,B 0,C 180,E1 -2688.675,E2 -2688.675} C_VEL
LIN {X 0,Y 566.208,Z 400.958,A -85,B 0,C 180,E1 -2691.434,E2 -2691.434} C_VEL
LIN {X 0,Y 566.263,Z 400.951,A -85,B 0,C 180,E1 -2694.302,E2 -2694.302} C_VEL
LIN {X 0,Y 566.288,Z 400.949,A -85,B 0,C 180,E1 -2697.866,E2 -2697.866} C_VEL
LIN {X 0,Y 566.308,Z 400.944,A -85,B 0,C 180,E1 -2700.711,E2 -2700.711} C_VEL
LIN {X 0,Y 566.276,Z 400.948,A -85,B 0,C 180,E1 -2702.846,E2 -2702.846} C_VEL
LIN {X 0,Y 566.259,Z 400.953,A -85,B 0,C 180,E1 -2705.698,E2 -2705.698} C_VEL
LIN {X 0,Y 566.237,Z 400.954,A -85,B 0,C 180,E1 -2708.566,E2 -2708.566} C_VEL
LIN {X 0,Y 566.245,Z 400.953,A -85,B 0,C 180,E1 -2711.454,E2 -2711.454} C_VEL
LIN {X 0,Y 566.237,Z 400.954,A -85,B 0,C 180,E1 -2714.507,E2 -2714.507} C_VEL
LIN {X 0,Y 566.203,Z 400.958,A -85,B 0,C 180,E1 -2717.332,E2 -2717.332} C_VEL
LIN {X 0,Y 566.223,Z 400.956,A -85,B 0,C 180,E1 -2720.337,E2 -2720.337} C_VEL
LIN {X 0,Y 566.193,Z 400.959,A -85,B 0,C 180,E1 -2723.404,E2 -2723.404} C_VEL
LIN {X 0,Y 566.217,Z 400.956,A -85,B 0,C 180,E1 -2725.749,E2 -2725.749} C_VEL
LIN {X 0,Y 566.206,Z 400.959,A -85,B 0,C 180,E1 -2727.488,E2 -2727.488} C_VEL
LIN {X 0,Y 565.526,Z 401.044,A -85,B 0,C 180,E1 -2728.082,E2 -2728.082} C_VEL
LIN {X 0,Y 562.66,Z 401.398,A -85,B 0,C 180,E1 -2729.045,E2 -2729.045} C_VEL
LIN {X 0,Y 560.25,Z 401.7,A -85,B 0,C 180,E1 -2729.821,E2 -2729.821} C_VEL
LIN {X 0,Y 559.222,Z 401.83,A -85,B 0,C 180,E1 -2730.42,E2 -2730.42} C_VEL
LIN {X 0,Y 559.142,Z 401.836,A -85,B 0,C 180,E1 -2730.622,E2 -2730.622} C_VEL
LIN {X 0,Y 559.168,Z 401.835,A -85,B 0,C 180,E1 -2733.575,E2 -2733.575} C_VEL
LIN {X 0,Y 559.171,Z 401.834,A -85,B 0,C 180,E1 -2736.449,E2 -2736.449} C_VEL
LIN {X 0,Y 559.177,Z 401.833,A -85,B 0,C 180,E1 -2738.934,E2 -2738.934} C_VEL
LIN {X 0,Y 559.18,Z 401.833,A -85,B 0,C 180,E1 -2742.138,E2 -2742.138} C_VEL
LIN {X 0,Y 559.144,Z 401.838,A -85,B 0,C 180,E1 -2744.739,E2 -2744.739} C_VEL
LIN {X 0,Y 559.168,Z 401.834,A -85,B 0,C 180,E1 -2747.257,E2 -2747.257} C_VEL
LIN {X 0,Y 559.185,Z 401.834,A -85,B 0,C 180,E1 -2750.135,E2 -2750.135} C_VEL
LIN {X 0,Y 559.147,Z 401.836,A -85,B 0,C 180,E1 -2752.892,E2 -2752.892} C_VEL
LIN {X 0,Y 559.162,Z 401.837,A -85,B 0,C 180,E1 -2755.556,E2 -2755.556} C_VEL
LIN {X 0,Y 559.177,Z 401.833,A -85,B 0,C 180,E1 -2758.138,E2 -2758.138} C_VEL
LIN {X 0,Y 559.162,Z 401.836,A -85,B 0,C 180,E1 -2760.647,E2 -2760.647} C_VEL
LIN {X 0,Y 559.175,Z 401.835,A -85,B 0,C 180,E1 -2763.173,E2 -2763.173} C_VEL
LIN {X 0,Y 559.162,Z 401.836,A -85,B 0,C 180,E1 -2765.495,E2 -2765.495} C_VEL
LIN {X 0,Y 559.177,Z 401.834,A -85,B 0,C 180,E1 -2768.624,E2 -2768.624} C_VEL
LIN {X 0,Y 559.174,Z 401.834,A -85,B 0,C 180,E1 -2770.927,E2 -2770.927} C_VEL
LIN {X 0,Y 559.168,Z 401.836,A -85,B 0,C 180,E1 -2773.948,E2 -2773.948} C_VEL
LIN {X 0,Y 559.176,Z 401.835,A -85,B 0,C 180,E1 -2776.184,E2 -2776.184} C_VEL
LIN {X 0,Y 559.201,Z 401.832,A -85,B 0,C 180,E1 -2779.134,E2 -2779.134} C_VEL
LIN {X 0,Y 559.209,Z 401.83,A -85,B 0,C 180,E1 -2780.848,E2 -2780.848} C_VEL
LIN {X 0,Y 559.79,Z 405.749,A -85,B 0,C 180,E1 -2781.017,E2 -2781.017} C_VEL
LIN {X 0,Y 559.631,Z 418.038,A -85,B 0,C 180,E1 -2781.606,E2 -2781.606} C_VEL
LIN {X 0,Y 559.473,Z 428.292,A -85,B 0,C 180,E1 -2782.239,E2 -2782.239} C_VEL
LIN {X 0,Y 559.333,Z 437.395,A -85,B 0,C 180,E1 -2782.921,E2 -2782.921} C_VEL
LIN {X 0,Y 559.164,Z 445.996,A -85,B 0,C 180,E1 -2783.686,E2 -2783.686} C_VEL
LIN {X 0,Y 559.141,Z 454.262,A -85,B 0,C 180,E1 -2784.591,E2 -2784.591} C_VEL
LIN {X 0,Y 559.015,Z 462.472,A -85,B 0,C 180,E1 -2785.674,E2 -2785.674} C_VEL
LIN {X 0,Y 558.927,Z 469.049,A -85,B 0,C 180,E1 -2786.756,E2 -2786.756} C_VEL
LIN {X 0,Y 558.793,Z 474.285,A -85,B 0,C 180,E1 -2787.838,E2 -2787.838} C_VEL
LIN {X 0,Y 558.818,Z 478.371,A -85,B 0,C 180,E1 -2788.919,E2 -2788.919} C_VEL
LIN {X 0,Y 558.745,Z 481.419,A -85,B 0,C 180,E1 -2790,E2 -2790} C_VEL
LIN {X 0,Y 558.742,Z 482.922,A -85,B 0,C 180,E1 -2790.721,E2 -2790.721} C_VEL
LIN {X 0,Y 558.745,Z 484.682,A -85,B 0,C 180,E1 -2792.163,E2 -2792.163} C_VEL
LIN {X 0,Y 558.82,Z 484.88,A -85,B 0,C 180,E1 -2793.605,E2 -2793.605} C_VEL
LIN {X 0,Y 558.766,Z 483.445,A -85,B 0,C 180,E1 -2795.051,E2 -2795.051} C_VEL
LIN {X 0,Y 558.848,Z 480.281,A -85,B 0,C 180,E1 -2796.536,E2 -2796.536} C_VEL
LIN {X 0,Y 558.826,Z 476.919,A -85,B 0,C 180,E1 -2797.588,E2 -2797.588} C_VEL
LIN {X 0,Y 558.87,Z 472.319,A -85,B 0,C 180,E1 -2798.68,E2 -2798.68} C_VEL
LIN {X 0,Y 558.948,Z 466.491,A -85,B 0,C 180,E1 -2799.773,E2 -2799.773} C_VEL
LIN {X 0,Y 558.981,Z 460.603,A -85,B 0,C 180,E1 -2800.688,E2 -2800.688} C_VEL
LIN {X 0,Y 559.099,Z 453.376,A -85,B 0,C 180,E1 -2801.603,E2 -2801.603} C_VEL
LIN {X 0,Y 559.225,Z 444.766,A -85,B 0,C 180,E1 -2802.521,E2 -2802.521} C_VEL
LIN {X 0,Y 559.358,Z 434.057,A -85,B 0,C 180,E1 -2803.441,E2 -2803.441} C_VEL
LIN {X 0,Y 559.551,Z 423.332,A -85,B 0,C 180,E1 -2804.177,E2 -2804.177} C_VEL
LIN {X 0,Y 559.731,Z 411.868,A -85,B 0,C 180,E1 -2804.8,E2 -2804.8} C_VEL
LIN {X 0,Y 559.687,Z 403.868,A -85,B 0,C 180,E1 -2805.151,E2 -2805.151} C_VEL
LIN {X 0,Y 559.225,Z 401.826,A -85,B 0,C 180,E1 -2805.263,E2 -2805.263} C_VEL
LIN {X 0,Y 559.147,Z 401.839,A -85,B 0,C 180,E1 -2808.314,E2 -2808.314} C_VEL
LIN {X 0,Y 559.182,Z 401.832,A -85,B 0,C 180,E1 -2810.605,E2 -2810.605} C_VEL
LIN {X 0,Y 559.141,Z 401.832,A -85,B 0,C 180,E1 -2813.717,E2 -2813.717} C_VEL
LIN {X 0,Y 559.184,Z 401.831,A -85,B 0,C 180,E1 -2816.097,E2 -2816.097} C_VEL
LIN {X 0,Y 559.168,Z 401.833,A -85,B 0,C 180,E1 -2818.53,E2 -2818.53} C_VEL
LIN {X 0,Y 559.151,Z 401.829,A -85,B 0,C 180,E1 -2821.273,E2 -2821.273} C_VEL
LIN {X 0,Y 559.173,Z 401.832,A -85,B 0,C 180,E1 -2823.949,E2 -2823.949} C_VEL
LIN {X 0,Y 559.149,Z 401.829,A -85,B 0,C 180,E1 -2827.108,E2 -2827.108} C_VEL
LIN {X 0,Y 559.167,Z 401.834,A -85,B 0,C 180,E1 -2829.942,E2 -2829.942} C_VEL
LIN {X 0,Y 559.162,Z 401.829,A -85,B 0,C 180,E1 -2832.744,E2 -2832.744} C_VEL
LIN {X 0,Y 559.161,Z 401.833,A -85,B 0,C 180,E1 -2835.76,E2 -2835.76} C_VEL
LIN {X 0,Y 559.194,Z 401.83,A -85,B 0,C 180,E1 -2838.232,E2 -2838.232} C_VEL
LIN {X 0,Y 559.179,Z 401.826,A -85,B 0,C 180,E1 -2841.192,E2 -2841.192} C_VEL
LIN {X 0,Y 559.144,Z 401.837,A -85,B 0,C 180,E1 -2843.789,E2 -2843.789} C_VEL
LIN {X 0,Y 559.168,Z 401.83,A -85,B 0,C 180,E1 -2846.425,E2 -2846.425} C_VEL
LIN {X 0,Y 559.16,Z 401.828,A -85,B 0,C 180,E1 -2848.981,E2 -2848.981} C_VEL
LIN {X 0,Y 559.173,Z 401.832,A -85,B 0,C 180,E1 -2851.619,E2 -2851.619} C_VEL
LIN {X 0,Y 559.181,Z 401.825,A -85,B 0,C 180,E1 -2854.702,E2 -2854.702} C_VEL
LIN {X 0,Y 559.146,Z 401.839,A -85,B 0,C 180,E1 -2857.847,E2 -2857.847} C_VEL
LIN {X 0,Y 559.198,Z 401.824,A -85,B 0,C 180,E1 -2860.494,E2 -2860.494} C_VEL
LIN {X 0,Y 559.184,Z 401.827,A -85,B 0,C 180,E1 -2863.197,E2 -2863.197} C_VEL
LIN {X 0,Y 559.175,Z 401.83,A -85,B 0,C 180,E1 -2866.184,E2 -2866.184} C_VEL
LIN {X 0,Y 559.202,Z 401.949,A -85,B 0,C 180,E1 -2868.858,E2 -2868.858} C_VEL
LIN {X 0,Y 559.807,Z 404.833,A -85,B 0,C 180,E1 -2868.979,E2 -2868.979} C_VEL
LIN {X 0,Y 559.697,Z 416.202,A -85,B 0,C 180,E1 -2869.509,E2 -2869.509} C_VEL
LIN {X 0,Y 559.537,Z 425.55,A -85,B 0,C 180,E1 -2870.055,E2 -2870.055} C_VEL
LIN {X 0,Y 559.366,Z 435.672,A -85,B 0,C 180,E1 -2870.782,E2 -2870.782} C_VEL
LIN {X 0,Y 559.269,Z 444.054,A -85,B 0,C 180,E1 -2871.509,E2 -2871.509} C_VEL
LIN {X 0,Y 559.098,Z 452.77,A -85,B 0,C 180,E1 -2872.415,E2 -2872.415} C_VEL
LIN {X 0,Y 558.987,Z 461.313,A -85,B 0,C 180,E1 -2873.503,E2 -2873.503} C_VEL
LIN {X 0,Y 558.885,Z 468.106,A -85,B 0,C 180,E1 -2874.588,E2 -2874.588} C_VEL
LIN {X 0,Y 558.899,Z 473.526,A -85,B 0,C 180,E1 -2875.673,E2 -2875.673} C_VEL
LIN {X 0,Y 558.856,Z 477.775,A -85,B 0,C 180,E1 -2876.756,E2 -2876.756} C_VEL
LIN {X 0,Y 558.764,Z 480.98,A -85,B 0,C 180,E1 -2877.837,E2 -2877.837} C_VEL
LIN {X 0,Y 558.749,Z 482.625,A -85,B 0,C 180,E1 -2878.558,E2 -2878.558} C_VEL
LIN {X 0,Y 558.742,Z 483.793,A -85,B 0,C 180,E1 -2879.279,E2 -2879.279} C_VEL
LIN {X 0,Y 558.74,Z 484.94,A -85,B 0,C 180,E1 -2880.721,E2 -2880.721} C_VEL
LIN {X 0,Y 558.745,Z 484.924,A -85,B 0,C 180,E1 -2881.441,E2 -2881.441} C_VEL
LIN {X 0,Y 558.795,Z 483.682,A -85,B 0,C 180,E1 -2882.884,E2 -2882.884} C_VEL
LIN {X 0,Y 558.825,Z 482.481,A -85,B 0,C 180,E1 -2883.605,E2 -2883.605} C_VEL
LIN {X 0,Y 558.788,Z 478.728,A -85,B 0,C 180,E1 -2885.051,E2 -2885.051} C_VEL
LIN {X 0,Y 558.878,Z 475.126,A -85,B 0,C 180,E1 -2886.043,E2 -2886.043} C_VEL
LIN {X 0,Y 558.905,Z 469.58,A -85,B 0,C 180,E1 -2887.224,E2 -2887.224} C_VEL
LIN {X 0,Y 558.992,Z 463.131,A -85,B 0,C 180,E1 -2888.313,E2 -2888.313} C_VEL
LIN {X 0,Y 559.065,Z 455.104,A -85,B 0,C 180,E1 -2889.406,E2 -2889.406} C_VEL
LIN {X 0,Y 559.227,Z 446.848,A -85,B 0,C 180,E1 -2890.316,E2 -2890.316} C_VEL
LIN {X 0,Y 559.336,Z 436.954,A -85,B 0,C 180,E1 -2891.206,E2 -2891.206} C_VEL
LIN {X 0,Y 559.514,Z 428.011,A -85,B 0,C 180,E1 -2891.87,E2 -2891.87} C_VEL
LIN {X 0,Y 559.602,Z 419.115,A -85,B 0,C 180,E1 -2892.42,E2 -2892.42} C_VEL
LIN {X 0,Y 559.736,Z 409.094,A -85,B 0,C 180,E1 -2892.924,E2 -2892.924} C_VEL
LIN {X 0,Y 559.608,Z 403.784,A -85,B 0,C 180,E1 -2893.157,E2 -2893.157} C_VEL
LIN {X 0,Y 559.173,Z 401.837,A -85,B 0,C 180,E1 -2893.237,E2 -2893.237} C_VEL
LIN {X 0,Y 559.154,Z 401.835,A -85,B 0,C 180,E1 -2895.304,E2 -2895.304} C_VEL
LIN {X 0,Y 559.146,Z 401.841,A -85,B 0,C 180,E1 -2897.557,E2 -2897.557} C_VEL
LIN {X 0,Y 559.177,Z 401.834,A -85,B 0,C 180,E1 -2899.837,E2 -2899.837} C_VEL
LIN {X 0,Y 559.146,Z 401.836,A -85,B 0,C 180,E1 -2902.153,E2 -2902.153} C_VEL
LIN {X 0,Y 559.181,Z 401.831,A -85,B 0,C 180,E1 -2905.298,E2 -2905.298} C_VEL
LIN {X 0,Y 559.186,Z 401.83,A -85,B 0,C 180,E1 -2907.712,E2 -2907.712} C_VEL
LIN {X 0,Y 559.158,Z 401.836,A -85,B 0,C 180,E1 -2910.183,E2 -2910.183} C_VEL
LIN {X 0,Y 559.161,Z 401.838,A -85,B 0,C 180,E1 -2912.715,E2 -2912.715} C_VEL
LIN {X 0,Y 559.131,Z 401.839,A -85,B 0,C 180,E1 -2915.324,E2 -2915.324} C_VEL
LIN {X 0,Y 559.135,Z 401.838,A -85,B 0,C 180,E1 -2918.018,E2 -2918.018} C_VEL
LIN {X 0,Y 559.16,Z 401.835,A -85,B 0,C 180,E1 -2920.812,E2 -2920.812} C_VEL
LIN {X 0,Y 559.167,Z 401.836,A -85,B 0,C 180,E1 -2923.732,E2 -2923.732} C_VEL
LIN {X 0,Y 559.149,Z 401.839,A -85,B 0,C 180,E1 -2926.803,E2 -2926.803} C_VEL
LIN {X 0,Y 559.177,Z 401.834,A -85,B 0,C 180,E1 -2929.189,E2 -2929.189} C_VEL
LIN {X 0,Y 559.139,Z 401.84,A -85,B 0,C 180,E1 -2931.983,E2 -2931.983} C_VEL
LIN {X 0,Y 559.197,Z 401.895,A -85,B 0,C 180,E1 -2932.94,E2 -2932.94} C_VEL
LIN {X 0,Y 560.154,Z 407.852,A -85,B 0,C 180,E1 -2934.291,E2 -2934.291} C_VEL
LIN {X 0,Y 560.029,Z 420.386,A -85,B 0,C 180,E1 -2936.902,E2 -2936.902} C_VEL
LIN {X 0,Y 559.971,Z 435.271,A -85,B 0,C 180,E1 -2939.866,E2 -2939.866} C_VEL
LIN {X 0,Y 559.905,Z 449.968,A -85,B 0,C 180,E1 -2942.718,E2 -2942.718} C_VEL
LIN {X 0,Y 559.839,Z 464.896,A -85,B 0,C 180,E1 -2945.526,E2 -2945.526} C_VEL
LIN {X 0,Y 559.742,Z 475.144,A -85,B 0,C 180,E1 -2947.483,E2 -2947.483} C_VEL
LIN {X 0,Y 559.522,Z 489.989,A -85,B 0,C 180,E1 -2950.4,E2 -2950.4} C_VEL
LIN {X 0,Y 559.323,Z 504.491,A -85,B 0,C 180,E1 -2953.202,E2 -2953.202} C_VEL
LIN {X 0,Y 559.175,Z 520.142,A -85,B 0,C 180,E1 -2956.184,E2 -2956.184} C_VEL
LIN {X 0,Y 559.103,Z 525.155,A -85,B 0,C 180,E1 -2957.131,E2 -2957.131} C_VEL
LIN {X 0,Y 560.028,Z 532.077,A -85,B 0,C 180,E1 -2957.267,E2 -2957.267} C_VEL
LIN {X 0,Y 559.911,Z 545.733,A -85,B 0,C 180,E1 -2957.61,E2 -2957.61} C_VEL
LIN {X 0,Y 559.803,Z 557.49,A -85,B 0,C 180,E1 -2958.045,E2 -2958.045} C_VEL
LIN {X 0,Y 559.636,Z 569.832,A -85,B 0,C 180,E1 -2958.662,E2 -2958.662} C_VEL
LIN {X 0,Y 559.434,Z 581.48,A -85,B 0,C 180,E1 -2959.413,E2 -2959.413} C_VEL
LIN {X 0,Y 559.297,Z 591.645,A -85,B 0,C 180,E1 -2960.233,E2 -2960.233} C_VEL
LIN {X 0,Y 559.134,Z 600.785,A -85,B 0,C 180,E1 -2961.142,E2 -2961.142} C_VEL
LIN {X 0,Y 559.01,Z 609.688,A -85,B 0,C 180,E1 -2962.232,E2 -2962.232} C_VEL
LIN {X 0,Y 558.925,Z 615.74,A -85,B 0,C 180,E1 -2963.14,E2 -2963.14} C_VEL
LIN {X 0,Y 558.935,Z 621.679,A -85,B 0,C 180,E1 -2964.227,E2 -2964.227} C_VEL
LIN {X 0,Y 558.827,Z 626.371,A -85,B 0,C 180,E1 -2965.311,E2 -2965.311} C_VEL
LIN {X 0,Y 558.836,Z 629.957,A -85,B 0,C 180,E1 -2966.395,E2 -2966.395} C_VEL
LIN {X 0,Y 558.799,Z 631.808,A -85,B 0,C 180,E1 -2967.116,E2 -2967.116} C_VEL
LIN {X 0,Y 558.745,Z 634.185,A -85,B 0,C 180,E1 -2968.558,E2 -2968.558} C_VEL
LIN {X 0,Y 558.74,Z 635,A -85,B 0,C 180,E1 -2970,E2 -2970} C_VEL
LIN {X 0,Y 558.745,Z 634.186,A -85,B 0,C 180,E1 -2971.441,E2 -2971.441} C_VEL
LIN {X 0,Y 558.799,Z 631.81,A -85,B 0,C 180,E1 -2972.883,E2 -2972.883} C_VEL
LIN {X 0,Y 558.843,Z 628.896,A -85,B 0,C 180,E1 -2973.966,E2 -2973.966} C_VEL
LIN {X 0,Y 558.799,Z 624.949,A -85,B 0,C 180,E1 -2975.051,E2 -2975.051} C_VEL
LIN {X 0,Y 558.921,Z 619.868,A -85,B 0,C 180,E1 -2976.135,E2 -2976.135} C_VEL
LIN {X 0,Y 558.977,Z 613.469,A -85,B 0,C 180,E1 -2977.223,E2 -2977.223} C_VEL
LIN {X 0,Y 559.099,Z 605.479,A -85,B 0,C 180,E1 -2978.312,E2 -2978.312} C_VEL
LIN {X 0,Y 559.195,Z 597.336,A -85,B 0,C 180,E1 -2979.221,E2 -2979.221} C_VEL
LIN {X 0,Y 559.351,Z 587.402,A -85,B 0,C 180,E1 -2980.131,E2 -2980.131} C_VEL
LIN {X 0,Y 559.533,Z 576.4,A -85,B 0,C 180,E1 -2980.937,E2 -2980.937} C_VEL
LIN {X 0,Y 559.671,Z 564.464,A -85,B 0,C 180,E1 -2981.628,E2 -2981.628} C_VEL
LIN {X 0,Y 559.806,Z 551.77,A -85,B 0,C 180,E1 -2982.185,E2 -2982.185} C_VEL
LIN {X 0,Y 559.989,Z 538.352,A -85,B 0,C 180,E1 -2982.595,E2 -2982.595} C_VEL
LIN {X 0,Y 559.822,Z 529.617,A -85,B 0,C 180,E1 -2982.783,E2 -2982.783} C_VEL
LIN {X 0,Y 559.112,Z 525.035,A -85,B 0,C 180,E1 -2982.892,E2 -2982.892} C_VEL
LIN {X 0,Y 559.252,Z 510.362,A -85,B 0,C 180,E1 -2985.675,E2 -2985.675} C_VEL
LIN {X 0,Y 559.427,Z 496.667,A -85,B 0,C 180,E1 -2988.305,E2 -2988.305} C_VEL
LIN {X 0,Y 559.626,Z 482.972,A -85,B 0,C 180,E1 -2990.972,E2 -2990.972} C_VEL
LIN {X 0,Y 559.825,Z 469.113,A -85,B 0,C 180,E1 -2993.686,E2 -2993.686} C_VEL
LIN {X 0,Y 559.908,Z 454.28,A -85,B 0,C 180,E1 -2996.462,E2 -2996.462} C_VEL
LIN {X 0,Y 559.956,Z 439.491,A -85,B 0,C 180,E1 -2999.307,E2 -2999.307} C_VEL
LIN {X 0,Y 560.014,Z 424.756,A -85,B 0,C 180,E1 -3002.233,E2 -3002.233} C_VEL
LIN {X 0,Y 560.21,Z 409.489,A -85,B 0,C 180,E1 -3005.368,E2 -3005.368} C_VEL
LIN {X 0,Y 559.972,Z 405.882,A -85,B 0,C 180,E1 -3006.148,E2 -3006.148} C_VEL
LIN {X 0,Y 559.202,Z 401.832,A -85,B 0,C 180,E1 -3007.104,E2 -3007.104} C_VEL
LIN {X 0,Y 559.172,Z 401.834,A -85,B 0,C 180,E1 -3009.943,E2 -3009.943} C_VEL
LIN {X 0,Y 559.159,Z 401.837,A -85,B 0,C 180,E1 -3012.744,E2 -3012.744} C_VEL
LIN {X 0,Y 559.157,Z 401.838,A -85,B 0,C 180,E1 -3015.76,E2 -3015.76} C_VEL
LIN {X 0,Y 559.194,Z 401.832,A -85,B 0,C 180,E1 -3018.232,E2 -3018.232} C_VEL
LIN {X 0,Y 559.181,Z 401.834,A -85,B 0,C 180,E1 -3021.191,E2 -3021.191} C_VEL
LIN {X 0,Y 559.162,Z 401.835,A -85,B 0,C 180,E1 -3023.791,E2 -3023.791} C_VEL
LIN {X 0,Y 559.164,Z 401.836,A -85,B 0,C 180,E1 -3026.425,E2 -3026.425} C_VEL
LIN {X 0,Y 559.158,Z 401.836,A -85,B 0,C 180,E1 -3028.981,E2 -3028.981} C_VEL
LIN {X 0,Y 559.172,Z 401.833,A -85,B 0,C 180,E1 -3031.618,E2 -3031.618} C_VEL
LIN {X 0,Y 559.202,Z 401.83,A -85,B 0,C 180,E1 -3033.904,E2 -3033.904} C_VEL
LIN {X 0,Y 559.159,Z 401.836,A -85,B 0,C 180,E1 -3036.567,E2 -3036.567} C_VEL
LIN {X 0,Y 559.182,Z 401.833,A -85,B 0,C 180,E1 -3039.396,E2 -3039.396} C_VEL
LIN {X 0,Y 559.149,Z 401.838,A -85,B 0,C 180,E1 -3041.686,E2 -3041.686} C_VEL
LIN {X 0,Y 559.172,Z 401.836,A -85,B 0,C 180,E1 -3043.948,E2 -3043.948} C_VEL
LIN {X 0,Y 559.177,Z 401.835,A -85,B 0,C 180,E1 -3046.184,E2 -3046.184} C_VEL
LIN {X 0,Y 559.197,Z 401.831,A -85,B 0,C 180,E1 -3049.134,E2 -3049.134} C_VEL
LIN {X 0,Y 559.197,Z 401.831,A -85,B 0,C 180,E1 -3052.054,E2 -3052.054} C_VEL
LIN {X 0,Y 559.259,Z 401.824,A -85,B 0,C 180,E1 -3054.953,E2 -3054.953} C_VEL
LIN {X 0,Y 559.259,Z 401.824,A -85,B 0,C 180,E1 -3057.84,E2 -3057.84} C_VEL
LIN {X 0,Y 559.278,Z 401.82,A -85,B 0,C 180,E1 -3060.72,E2 -3060.72} C_VEL
LIN {X 0,Y 559.242,Z 401.824,A -85,B 0,C 180,E1 -3062.881,E2 -3062.881} C_VEL
LIN {X 0,Y 559.229,Z 401.828,A -85,B 0,C 180,E1 -3065.77,E2 -3065.77} C_VEL
LIN {X 0,Y 559.196,Z 401.832,A -85,B 0,C 180,E1 -3068.674,E2 -3068.674} C_VEL
LIN {X 0,Y 559.208,Z 401.829,A -85,B 0,C 180,E1 -3071.601,E2 -3071.601} C_VEL
LIN {X 0,Y 559.203,Z 401.83,A -85,B 0,C 180,E1 -3074.596,E2 -3074.596} C_VEL
LIN {X 0,Y 559.162,Z 401.837,A -85,B 0,C 180,E1 -3077.557,E2 -3077.557} C_VEL
LIN {X 0,Y 559.176,Z 401.835,A -85,B 0,C 180,E1 -3079.837,E2 -3079.837} C_VEL
LIN {X 0,Y 559.146,Z 401.838,A -85,B 0,C 180,E1 -3082.153,E2 -3082.153} C_VEL
LIN {X 0,Y 559.182,Z 401.834,A -85,B 0,C 180,E1 -3085.187,E2 -3085.187} C_VEL
LIN {X 0,Y 559.184,Z 401.833,A -85,B 0,C 180,E1 -3087.712,E2 -3087.712} C_VEL
LIN {X 0,Y 559.142,Z 401.836,A -85,B 0,C 180,E1 -3090.622,E2 -3090.622} C_VEL
LIN {X 0,Y 558.482,Z 401.92,A -85,B 0,C 180,E1 -3091.224,E2 -3091.224} C_VEL
LIN {X 0,Y 555.623,Z 402.276,A -85,B 0,C 180,E1 -3092.2,E2 -3092.2} C_VEL
LIN {X 0,Y 553.212,Z 402.577,A -85,B 0,C 180,E1 -3092.986,E2 -3092.986} C_VEL
LIN {X 0,Y 552.192,Z 402.704,A -85,B 0,C 180,E1 -3093.593,E2 -3093.593} C_VEL
LIN {X 0,Y 552.117,Z 402.711,A -85,B 0,C 180,E1 -3093.798,E2 -3093.798} C_VEL
LIN {X 0,Y 552.115,Z 402.713,A -85,B 0,C 180,E1 -3096.747,E2 -3096.747} C_VEL
LIN {X 0,Y 552.132,Z 402.711,A -85,B 0,C 180,E1 -3099.527,E2 -3099.527} C_VEL
LIN {X 0,Y 552.134,Z 402.712,A -85,B 0,C 180,E1 -3102.426,E2 -3102.426} C_VEL
LIN {X 0,Y 552.103,Z 402.716,A -85,B 0,C 180,E1 -3105.563,E2 -3105.563} C_VEL
LIN {X 0,Y 552.144,Z 402.71,A -85,B 0,C 180,E1 -3108.676,E2 -3108.676} C_VEL
LIN {X 0,Y 552.124,Z 402.713,A -85,B 0,C 180,E1 -3111.412,E2 -3111.412} C_VEL
LIN {X 0,Y 552.109,Z 402.715,A -85,B 0,C 180,E1 -3114.158,E2 -3114.158} C_VEL
LIN {X 0,Y 552.128,Z 402.711,A -85,B 0,C 180,E1 -3116.815,E2 -3116.815} C_VEL
LIN {X 0,Y 552.119,Z 402.712,A -85,B 0,C 180,E1 -3119.392,E2 -3119.392} C_VEL
LIN {X 0,Y 552.124,Z 402.714,A -85,B 0,C 180,E1 -3121.903,E2 -3121.903} C_VEL
LIN {X 0,Y 552.16,Z 402.706,A -85,B 0,C 180,E1 -3124.65,E2 -3124.65} C_VEL
LIN {X 0,Y 552.098,Z 402.716,A -85,B 0,C 180,E1 -3127.549,E2 -3127.549} C_VEL
LIN {X 0,Y 552.154,Z 402.709,A -85,B 0,C 180,E1 -3130.374,E2 -3130.374} C_VEL
LIN {X 0,Y 552.16,Z 402.708,A -85,B 0,C 180,E1 -3132.978,E2 -3132.978} C_VEL
LIN {X 0,Y 552.14,Z 402.712,A -85,B 0,C 180,E1 -3136.005,E2 -3136.005} C_VEL
LIN {X 0,Y 552.169,Z 402.707,A -85,B 0,C 180,E1 -3138.994,E2 -3138.994} C_VEL
LIN {X 0,Y 552.149,Z 402.714,A -85,B 0,C 180,E1 -3140.73,E2 -3140.73} C_VEL
LIN {X 0,Y 552.847,Z 406.66,A -85,B 0,C 180,E1 -3140.903,E2 -3140.903} C_VEL
LIN {X 0,Y 552.644,Z 418.757,A -85,B 0,C 180,E1 -3141.499,E2 -3141.499} C_VEL
LIN {X 0,Y 552.482,Z 428.841,A -85,B 0,C 180,E1 -3142.14,E2 -3142.14} C_VEL
LIN {X 0,Y 552.327,Z 438.109,A -85,B 0,C 180,E1 -3142.852,E2 -3142.852} C_VEL
LIN {X 0,Y 552.135,Z 446.378,A -85,B 0,C 180,E1 -3143.605,E2 -3143.605} C_VEL
LIN {X 0,Y 552.098,Z 454.586,A -85,B 0,C 180,E1 -3144.522,E2 -3144.522} C_VEL
LIN {X 0,Y 551.95,Z 462.739,A -85,B 0,C 180,E1 -3145.619,E2 -3145.619} C_VEL
LIN {X 0,Y 551.847,Z 469.256,A -85,B 0,C 180,E1 -3146.715,E2 -3146.715} C_VEL
LIN {X 0,Y 551.705,Z 474.433,A -85,B 0,C 180,E1 -3147.81,E2 -3147.81} C_VEL
LIN {X 0,Y 551.728,Z 478.494,A -85,B 0,C 180,E1 -3148.905,E2 -3148.905} C_VEL
LIN {X 0,Y 551.646,Z 481.493,A -85,B 0,C 180,E1 -3150,E2 -3150} C_VEL
LIN {X 0,Y 551.642,Z 482.997,A -85,B 0,C 180,E1 -3150.73,E2 -3150.73} C_VEL
LIN {X 0,Y 551.655,Z 484.707,A -85,B 0,C 180,E1 -3152.191,E2 -3152.191} C_VEL
LIN {X 0,Y 551.719,Z 484.98,A -85,B 0,C 180,E1 -3152.921,E2 -3152.921} C_VEL
LIN {X 0,Y 551.732,Z 484.86,A -85,B 0,C 180,E1 -3153.652,E2 -3153.652} C_VEL
LIN {X 0,Y 551.684,Z 483.387,A -85,B 0,C 180,E1 -3155.116,E2 -3155.116} C_VEL
LIN {X 0,Y 551.748,Z 480.273,A -85,B 0,C 180,E1 -3156.583,E2 -3156.583} C_VEL
LIN {X 0,Y 551.756,Z 476.772,A -85,B 0,C 180,E1 -3157.686,E2 -3157.686} C_VEL
LIN {X 0,Y 551.796,Z 472.118,A -85,B 0,C 180,E1 -3158.792,E2 -3158.792} C_VEL
LIN {X 0,Y 551.896,Z 466.245,A -85,B 0,C 180,E1 -3159.899,E2 -3159.899} C_VEL
LIN {X 0,Y 551.943,Z 460.329,A -85,B 0,C 180,E1 -3160.825,E2 -3160.825} C_VEL
LIN {X 0,Y 552.057,Z 453.025,A -85,B 0,C 180,E1 -3161.753,E2 -3161.753} C_VEL
LIN {X 0,Y 552.181,Z 444.343,A -85,B 0,C 180,E1 -3162.683,E2 -3162.683} C_VEL
LIN {X 0,Y 552.349,Z 433.552,A -85,B 0,C 180,E1 -3163.615,E2 -3163.615} C_VEL
LIN {X 0,Y 552.573,Z 422.644,A -85,B 0,C 180,E1 -3164.36,E2 -3164.36} C_VEL
LIN {X 0,Y 552.774,Z 410.344,A -85,B 0,C 180,E1 -3165.024,E2 -3165.024} C_VEL
LIN {X 0,Y 552.694,Z 404.977,A -85,B 0,C 180,E1 -3165.263,E2 -3165.263} C_VEL
LIN {X 0,Y 552.186,Z 402.703,A -85,B 0,C 180,E1 -3165.367,E2 -3165.367} C_VEL
LIN {X 0,Y 552.126,Z 402.713,A -85,B 0,C 180,E1 -3168.556,E2 -3168.556} C_VEL
LIN {X 0,Y 552.124,Z 402.708,A -85,B 0,C 180,E1 -3170.88,E2 -3170.88} C_VEL
LIN {X 0,Y 552.108,Z 402.712,A -85,B 0,C 180,E1 -3174.038,E2 -3174.038} C_VEL
LIN {X 0,Y 552.123,Z 402.712,A -85,B 0,C 180,E1 -3176.457,E2 -3176.457} C_VEL
LIN {X 0,Y 552.115,Z 402.707,A -85,B 0,C 180,E1 -3178.928,E2 -3178.928} C_VEL
LIN {X 0,Y 552.116,Z 402.706,A -85,B 0,C 180,E1 -3181.476,E2 -3181.476} C_VEL
LIN {X 0,Y 552.142,Z 402.712,A -85,B 0,C 180,E1 -3184.171,E2 -3184.171} C_VEL
LIN {X 0,Y 552.114,Z 402.707,A -85,B 0,C 180,E1 -3186.747,E2 -3186.747} C_VEL
LIN {X 0,Y 552.135,Z 402.704,A -85,B 0,C 180,E1 -3189.527,E2 -3189.527} C_VEL
LIN {X 0,Y 552.135,Z 402.708,A -85,B 0,C 180,E1 -3192.425,E2 -3192.425} C_VEL
LIN {X 0,Y 552.105,Z 402.709,A -85,B 0,C 180,E1 -3195.563,E2 -3195.563} C_VEL
LIN {X 0,Y 552.135,Z 402.704,A -85,B 0,C 180,E1 -3198.677,E2 -3198.677} C_VEL
LIN {X 0,Y 552.122,Z 402.706,A -85,B 0,C 180,E1 -3201.411,E2 -3201.411} C_VEL
LIN {X 0,Y 552.09,Z 402.715,A -85,B 0,C 180,E1 -3204.156,E2 -3204.156} C_VEL
LIN {X 0,Y 552.12,Z 402.705,A -85,B 0,C 180,E1 -3206.814,E2 -3206.814} C_VEL
LIN {X 0,Y 552.107,Z 402.709,A -85,B 0,C 180,E1 -3209.391,E2 -3209.391} C_VEL
LIN {X 0,Y 552.112,Z 402.715,A -85,B 0,C 180,E1 -3211.902,E2 -3211.902} C_VEL
LIN {X 0,Y 552.161,Z 402.7,A -85,B 0,C 180,E1 -3214.65,E2 -3214.65} C_VEL
LIN {X 0,Y 552.097,Z 402.714,A -85,B 0,C 180,E1 -3217.549,E2 -3217.549} C_VEL
LIN {X 0,Y 552.15,Z 402.703,A -85,B 0,C 180,E1 -3220.375,E2 -3220.375} C_VEL
LIN {X 0,Y 552.138,Z 402.703,A -85,B 0,C 180,E1 -3222.977,E2 -3222.977} C_VEL
LIN {X 0,Y 552.139,Z 402.709,A -85,B 0,C 180,E1 -3226.004,E2 -3226.004} C_VEL
LIN {X 0,Y 552.145,Z 402.705,A -85,B 0,C 180,E1 -3228.727,E2 -3228.727} C_VEL
LIN {X 0,Y 552.821,Z 406.86,A -85,B 0,C 180,E1 -3228.914,E2 -3228.914} C_VEL
LIN {X 0,Y 552.725,Z 416.427,A -85,B 0,C 180,E1 -3229.375,E2 -3229.375} C_VEL
LIN {X 0,Y 552.554,Z 425.735,A -85,B 0,C 180,E1 -3229.928,E2 -3229.928} C_VEL
LIN {X 0,Y 552.364,Z 434.695,A -85,B 0,C 180,E1 -3230.571,E2 -3230.571} C_VEL
LIN {X 0,Y 552.275,Z 442.27,A -85,B 0,C 180,E1 -3231.216,E2 -3231.216} C_VEL
LIN {X 0,Y 552.12,Z 449.637,A -85,B 0,C 180,E1 -3231.951,E2 -3231.951} C_VEL
LIN {X 0,Y 552.003,Z 457.342,A -85,B 0,C 180,E1 -3232.869,E2 -3232.869} C_VEL
LIN {X 0,Y 551.954,Z 463.768,A -85,B 0,C 180,E1 -3233.787,E2 -3233.787} C_VEL
LIN {X 0,Y 551.823,Z 468.176,A -85,B 0,C 180,E1 -3234.519,E2 -3234.519} C_VEL
LIN {X 0,Y 551.815,Z 473.575,A -85,B 0,C 180,E1 -3235.617,E2 -3235.617} C_VEL
LIN {X 0,Y 551.781,Z 477.814,A -85,B 0,C 180,E1 -3236.714,E2 -3236.714} C_VEL
LIN {X 0,Y 551.674,Z 481.007,A -85,B 0,C 180,E1 -3237.81,E2 -3237.81} C_VEL
LIN {X 0,Y 551.65,Z 482.645,A -85,B 0,C 180,E1 -3238.54,E2 -3238.54} C_VEL
LIN {X 0,Y 551.642,Z 483.812,A -85,B 0,C 180,E1 -3239.27,E2 -3239.27} C_VEL
LIN {X 0,Y 551.641,Z 484.939,A -85,B 0,C 180,E1 -3240.73,E2 -3240.73} C_VEL
LIN {X 0,Y 551.645,Z 484.922,A -85,B 0,C 180,E1 -3241.46,E2 -3241.46} C_VEL
LIN {X 0,Y 551.72,Z 483.66,A -85,B 0,C 180,E1 -3242.921,E2 -3242.921} C_VEL
LIN {X 0,Y 551.738,Z 482.457,A -85,B 0,C 180,E1 -3243.652,E2 -3243.652} C_VEL
LIN {X 0,Y 551.714,Z 478.677,A -85,B 0,C 180,E1 -3245.116,E2 -3245.116} C_VEL
LIN {X 0,Y 551.797,Z 476.176,A -85,B 0,C 180,E1 -3245.848,E2 -3245.848} C_VEL
LIN {X 0,Y 551.82,Z 471.407,A -85,B 0,C 180,E1 -3246.949,E2 -3246.949} C_VEL
LIN {X 0,Y 551.881,Z 465.349,A -85,B 0,C 180,E1 -3248.052,E2 -3248.052} C_VEL
LIN {X 0,Y 551.98,Z 459.193,A -85,B 0,C 180,E1 -3248.973,E2 -3248.973} C_VEL
LIN {X 0,Y 552.087,Z 451.789,A -85,B 0,C 180,E1 -3249.896,E2 -3249.896} C_VEL
LIN {X 0,Y 552.23,Z 444.771,A -85,B 0,C 180,E1 -3250.634,E2 -3250.634} C_VEL
LIN {X 0,Y 552.287,Z 436.508,A -85,B 0,C 180,E1 -3251.372,E2 -3251.372} C_VEL
LIN {X 0,Y 552.529,Z 427.796,A -85,B 0,C 180,E1 -3252.022,E2 -3252.022} C_VEL
LIN {X 0,Y 552.653,Z 418.856,A -85,B 0,C 180,E1 -3252.578,E2 -3252.578} C_VEL
LIN {X 0,Y 552.799,Z 408.776,A -85,B 0,C 180,E1 -3253.089,E2 -3253.089} C_VEL
LIN {X 0,Y 552.556,Z 404.595,A -85,B 0,C 180,E1 -3253.282,E2 -3253.282} C_VEL
LIN {X 0,Y 552.114,Z 402.715,A -85,B 0,C 180,E1 -3253.386,E2 -3253.386} C_VEL
LIN {X 0,Y 552.114,Z 402.712,A -85,B 0,C 180,E1 -3255.504,E2 -3255.504} C_VEL
LIN {X 0,Y 552.103,Z 402.716,A -85,B 0,C 180,E1 -3257.789,E2 -3257.789} C_VEL
LIN {X 0,Y 552.136,Z 402.714,A -85,B 0,C 180,E1 -3260.101,E2 -3260.101} C_VEL
LIN {X 0,Y 552.096,Z 402.715,A -85,B 0,C 180,E1 -3262.451,E2 -3262.451} C_VEL
LIN {X 0,Y 552.161,Z 402.706,A -85,B 0,C 180,E1 -3265.35,E2 -3265.35} C_VEL
LIN {X 0,Y 552.124,Z 402.71,A -85,B 0,C 180,E1 -3268.098,E2 -3268.098} C_VEL
LIN {X 0,Y 552.107,Z 402.712,A -85,B 0,C 180,E1 -3270.609,E2 -3270.609} C_VEL
LIN {X 0,Y 552.119,Z 402.71,A -85,B 0,C 180,E1 -3273.186,E2 -3273.186} C_VEL
LIN {X 0,Y 552.089,Z 402.716,A -85,B 0,C 180,E1 -3275.843,E2 -3275.843} C_VEL
LIN {X 0,Y 552.12,Z 402.712,A -85,B 0,C 180,E1 -3278.589,E2 -3278.589} C_VEL
LIN {X 0,Y 552.127,Z 402.71,A -85,B 0,C 180,E1 -3281.446,E2 -3281.446} C_VEL
LIN {X 0,Y 552.098,Z 402.713,A -85,B 0,C 180,E1 -3284.532,E2 -3284.532} C_VEL
LIN {X 0,Y 552.133,Z 402.71,A -85,B 0,C 180,E1 -3287.585,E2 -3287.585} C_VEL
LIN {X 0,Y 552.136,Z 402.711,A -85,B 0,C 180,E1 -3290.473,E2 -3290.473} C_VEL
LIN {X 0,Y 552.175,Z 402.901,A -85,B 0,C 180,E1 -3292.745,E2 -3292.745} C_VEL
LIN {X 0,Y 553.236,Z 409.379,A -85,B 0,C 180,E1 -3294.242,E2 -3294.242} C_VEL
LIN {X 0,Y 553.069,Z 422.424,A -85,B 0,C 180,E1 -3297.001,E2 -3297.001} C_VEL
LIN {X 0,Y 552.968,Z 437.468,A -85,B 0,C 180,E1 -3300.039,E2 -3300.039} C_VEL
LIN {X 0,Y 552.888,Z 451.807,A -85,B 0,C 180,E1 -3302.849,E2 -3302.849} C_VEL
LIN {X 0,Y 552.782,Z 466.177,A -85,B 0,C 180,E1 -3305.594,E2 -3305.594} C_VEL
LIN {X 0,Y 552.676,Z 479.947,A -85,B 0,C 180,E1 -3308.17,E2 -3308.17} C_VEL
LIN {X 0,Y 552.453,Z 494.708,A -85,B 0,C 180,E1 -3311.071,E2 -3311.071} C_VEL
LIN {X 0,Y 552.269,Z 508.403,A -85,B 0,C 180,E1 -3313.742,E2 -3313.742} C_VEL
LIN {X 0,Y 552.061,Z 524.055,A -85,B 0,C 180,E1 -3316.753,E2 -3316.753} C_VEL
LIN {X 0,Y 552.072,Z 525.155,A -85,B 0,C 180,E1 -3316.964,E2 -3316.964} C_VEL
LIN {X 0,Y 553.111,Z 533.218,A -85,B 0,C 180,E1 -3317.129,E2 -3317.129} C_VEL
LIN {X 0,Y 552.973,Z 546.493,A -85,B 0,C 180,E1 -3317.475,E2 -3317.475} C_VEL
LIN {X 0,Y 552.814,Z 558.509,A -85,B 0,C 180,E1 -3317.938,E2 -3317.938} C_VEL
LIN {X 0,Y 552.635,Z 570.815,A -85,B 0,C 180,E1 -3318.574,E2 -3318.574} C_VEL
LIN {X 0,Y 552.446,Z 581.481,A -85,B 0,C 180,E1 -3319.277,E2 -3319.277} C_VEL
LIN {X 0,Y 552.283,Z 591.644,A -85,B 0,C 180,E1 -3320.108,E2 -3320.108} C_VEL
LIN {X 0,Y 552.104,Z 600.784,A -85,B 0,C 180,E1 -3321.029,E2 -3321.029} C_VEL
LIN {X 0,Y 551.96,Z 609.687,A -85,B 0,C 180,E1 -3322.133,E2 -3322.133} C_VEL
LIN {X 0,Y 551.835,Z 616.848,A -85,B 0,C 180,E1 -3323.234,E2 -3323.234} C_VEL
LIN {X 0,Y 551.804,Z 623.365,A -85,B 0,C 180,E1 -3324.518,E2 -3324.518} C_VEL
LIN {X 0,Y 551.764,Z 627.677,A -85,B 0,C 180,E1 -3325.617,E2 -3325.617} C_VEL
LIN {X 0,Y 551.75,Z 629.957,A -85,B 0,C 180,E1 -3326.348,E2 -3326.348} C_VEL
LIN {X 0,Y 551.723,Z 631.807,A -85,B 0,C 180,E1 -3327.079,E2 -3327.079} C_VEL
LIN {X 0,Y 551.645,Z 634.184,A -85,B 0,C 180,E1 -3328.54,E2 -3328.54} C_VEL
LIN {X 0,Y 551.64,Z 635,A -85,B 0,C 180,E1 -3330,E2 -3330} C_VEL
LIN {X 0,Y 551.645,Z 634.186,A -85,B 0,C 180,E1 -3331.46,E2 -3331.46} C_VEL
LIN {X 0,Y 551.723,Z 631.81,A -85,B 0,C 180,E1 -3332.921,E2 -3332.921} C_VEL
LIN {X 0,Y 551.763,Z 628.896,A -85,B 0,C 180,E1 -3334.017,E2 -3334.017} C_VEL
LIN {X 0,Y 551.724,Z 624.949,A -85,B 0,C 180,E1 -3335.116,E2 -3335.116} C_VEL
LIN {X 0,Y 551.803,Z 619.189,A -85,B 0,C 180,E1 -3336.341,E2 -3336.341} C_VEL
LIN {X 0,Y 551.926,Z 612.238,A -85,B 0,C 180,E1 -3337.499,E2 -3337.499} C_VEL
LIN {X 0,Y 552.082,Z 603.992,A -85,B 0,C 180,E1 -3338.602,E2 -3338.602} C_VEL
LIN {X 0,Y 552.201,Z 595.54,A -85,B 0,C 180,E1 -3339.523,E2 -3339.523} C_VEL
LIN {X 0,Y 552.419,Z 585.097,A -85,B 0,C 180,E1 -3340.445,E2 -3340.445} C_VEL
LIN {X 0,Y 552.599,Z 574.292,A -85,B 0,C 180,E1 -3341.213,E2 -3341.213} C_VEL
LIN {X 0,Y 552.781,Z 563.41,A -85,B 0,C 180,E1 -3341.83,E2 -3341.83} C_VEL
LIN {X 0,Y 552.88,Z 551.767,A -85,B 0,C 180,E1 -3342.34,E2 -3342.34} C_VEL
LIN {X 0,Y 553.067,Z 538.351,A -85,B 0,C 180,E1 -3342.755,E2 -3342.755} C_VEL
LIN {X 0,Y 552.912,Z 530.498,A -85,B 0,C 180,E1 -3342.931,E2 -3342.931} C_VEL
LIN {X 0,Y 552.058,Z 525.035,A -85,B 0,C 180,E1 -3343.06,E2 -3343.06} C_VEL
LIN {X 0,Y 552.225,Z 510.362,A -85,B 0,C 180,E1 -3345.88,E2 -3345.88} C_VEL
LIN {X 0,Y 552.434,Z 496.667,A -85,B 0,C 180,E1 -3348.545,E2 -3348.545} C_VEL
LIN {X 0,Y 552.654,Z 481.973,A -85,B 0,C 180,E1 -3351.445,E2 -3351.445} C_VEL
LIN {X 0,Y 552.793,Z 467.261,A -85,B 0,C 180,E1 -3354.206,E2 -3354.206} C_VEL
LIN {X 0,Y 552.867,Z 453.724,A -85,B 0,C 180,E1 -3356.785,E2 -3356.785} C_VEL
LIN {X 0,Y 553.002,Z 438.78,A -85,B 0,C 180,E1 -3359.712,E2 -3359.712} C_VEL
LIN {X 0,Y 553.038,Z 424.339,A -85,B 0,C 180,E1 -3362.625,E2 -3362.625} C_VEL
LIN {X 0,Y 553.283,Z 409.378,A -85,B 0,C 180,E1 -3365.754,E2 -3365.754} C_VEL
LIN {X 0,Y 552.133,Z 402.713,A -85,B 0,C 180,E1 -3367.316,E2 -3367.316} C_VEL
LIN {X 0,Y 552.144,Z 402.712,A -85,B 0,C 180,E1 -3370.478,E2 -3370.478} C_VEL
LIN {X 0,Y 552.093,Z 402.718,A -85,B 0,C 180,E1 -3373.481,E2 -3373.481} C_VEL
LIN {X 0,Y 552.122,Z 402.713,A -85,B 0,C 180,E1 -3376.578,E2 -3376.578} C_VEL
LIN {X 0,Y 552.124,Z 402.711,A -85,B 0,C 180,E1 -3379.52,E2 -3379.52} C_VEL
LIN {X 0,Y 552.096,Z 402.717,A -85,B 0,C 180,E1 -3382.336,E2 -3382.336} C_VEL
LIN {X 0,Y 552.121,Z 402.711,A -85,B 0,C 180,E1 -3385.054,E2 -3385.054} C_VEL
LIN {X 0,Y 552.117,Z 402.714,A -85,B 0,C 180,E1 -3387.681,E2 -3387.681} C_VEL
LIN {X 0,Y 552.114,Z 402.713,A -85,B 0,C 180,E1 -3390.235,E2 -3390.235} C_VEL
LIN {X 0,Y 552.15,Z 402.71,A -85,B 0,C 180,E1 -3392.998,E2 -3392.998} C_VEL
LIN {X 0,Y 552.116,Z 402.714,A -85,B 0,C 180,E1 -3395.161,E2 -3395.161} C_VEL
LIN {X 0,Y 552.098,Z 402.717,A -85,B 0,C 180,E1 -3397.549,E2 -3397.549} C_VEL
LIN {X 0,Y 552.158,Z 402.709,A -85,B 0,C 180,E1 -3400.675,E2 -3400.675} C_VEL
LIN {X 0,Y 552.122,Z 402.712,A -85,B 0,C 180,E1 -3403.737,E2 -3403.737} C_VEL
LIN {X 0,Y 552.14,Z 402.711,A -85,B 0,C 180,E1 -3406.005,E2 -3406.005} C_VEL
LIN {X 0,Y 552.165,Z 402.706,A -85,B 0,C 180,E1 -3408.994,E2 -3408.994} C_VEL
LIN {X 0,Y 552.152,Z 402.709,A -85,B 0,C 180,E1 -3411.952,E2 -3411.952} C_VEL
LIN {X 0,Y 552.233,Z 402.699,A -85,B 0,C 180,E1 -3414.889,E2 -3414.889} C_VEL
LIN {X 0,Y 552.23,Z 402.699,A -85,B 0,C 180,E1 -3417.812,E2 -3417.812} C_VEL
LIN {X 0,Y 552.248,Z 402.696,A -85,B 0,C 180,E1 -3420.729,E2 -3420.729} C_VEL
LIN {X 0,Y 552.208,Z 402.7,A -85,B 0,C 180,E1 -3422.918,E2 -3422.918} C_VEL
LIN {X 0,Y 552.2,Z 402.704,A -85,B 0,C 180,E1 -3425.844,E2 -3425.844} C_VEL
LIN {X 0,Y 552.166,Z 402.708,A -85,B 0,C 180,E1 -3428.786,E2 -3428.786} C_VEL
LIN {X 0,Y 552.166,Z 402.707,A -85,B 0,C 180,E1 -3431.751,E2 -3431.751} C_VEL
LIN {X 0,Y 552.139,Z 402.709,A -85,B 0,C 180,E1 -3434.749,E2 -3434.749} C_VEL
LIN {X 0,Y 552.113,Z 402.714,A -85,B 0,C 180,E1 -3437.789,E2 -3437.789} C_VEL
LIN {X 0,Y 552.136,Z 402.71,A -85,B 0,C 180,E1 -3440.101,E2 -3440.101} C_VEL
LIN {X 0,Y 552.1,Z 402.715,A -85,B 0,C 180,E1 -3442.451,E2 -3442.451} C_VEL
LIN {X 0,Y 552.158,Z 402.709,A -85,B 0,C 180,E1 -3445.351,E2 -3445.351} C_VEL
LIN {X 0,Y 552.122,Z 402.713,A -85,B 0,C 180,E1 -3448.098,E2 -3448.098} C_VEL
LIN {X 0,Y 552.105,Z 402.715,A -85,B 0,C 180,E1 -3450.619,E2 -3450.619} C_VEL
LIN {X 0,Y 552.126,Z 402.711,A -85,B 0,C 180,E1 -3453.185,E2 -3453.185} C_VEL
LIN {X 0,Y 552.117,Z 402.711,A -85,B 0,C 180,E1 -3453.798,E2 -3453.798} C_VEL
LIN {X 0,Y 551.481,Z 402.793,A -85,B 0,C 180,E1 -3454.407,E2 -3454.407} C_VEL
LIN {X 0,Y 548.659,Z 403.146,A -85,B 0,C 180,E1 -3455.395,E2 -3455.395} C_VEL
LIN {X 0,Y 546.239,Z 403.447,A -85,B 0,C 180,E1 -3456.19,E2 -3456.19} C_VEL
LIN {X 0,Y 545.17,Z 403.579,A -85,B 0,C 180,E1 -3456.804,E2 -3456.804} C_VEL
LIN {X 0,Y 545.068,Z 403.591,A -85,B 0,C 180,E1 -3457.012,E2 -3457.012} C_VEL
LIN {X 0,Y 545.069,Z 403.592,A -85,B 0,C 180,E1 -3460.143,E2 -3460.143} C_VEL
LIN {X 0,Y 545.09,Z 403.587,A -85,B 0,C 180,E1 -3463.106,E2 -3463.106} C_VEL
LIN {X 0,Y 545.068,Z 403.591,A -85,B 0,C 180,E1 -3466.225,E2 -3466.225} C_VEL
LIN {X 0,Y 545.101,Z 403.587,A -85,B 0,C 180,E1 -3468.887,E2 -3468.887} C_VEL
LIN {X 0,Y 545.057,Z 403.592,A -85,B 0,C 180,E1 -3471.763,E2 -3471.763} C_VEL
LIN {X 0,Y 545.062,Z 403.592,A -85,B 0,C 180,E1 -3474.534,E2 -3474.534} C_VEL
LIN {X 0,Y 545.087,Z 403.588,A -85,B 0,C 180,E1 -3477.213,E2 -3477.213} C_VEL
LIN {X 0,Y 545.107,Z 403.588,A -85,B 0,C 180,E1 -3479.813,E2 -3479.813} C_VEL
LIN {X 0,Y 545.097,Z 403.587,A -85,B 0,C 180,E1 -3482.827,E2 -3482.827} C_VEL
LIN {X 0,Y 545.055,Z 403.593,A -85,B 0,C 180,E1 -3485.631,E2 -3485.631} C_VEL
LIN {X 0,Y 545.071,Z 403.59,A -85,B 0,C 180,E1 -3488.837,E2 -3488.837} C_VEL
LIN {X 0,Y 545.087,Z 403.588,A -85,B 0,C 180,E1 -3491.196,E2 -3491.196} C_VEL
LIN {X 0,Y 545.076,Z 403.59,A -85,B 0,C 180,E1 -3493.521,E2 -3493.521} C_VEL
LIN {X 0,Y 545.1,Z 403.588,A -85,B 0,C 180,E1 -3495.82,E2 -3495.82} C_VEL
LIN {X 0,Y 545.124,Z 403.584,A -85,B 0,C 180,E1 -3498.85,E2 -3498.85} C_VEL
LIN {X 0,Y 545.125,Z 403.586,A -85,B 0,C 180,E1 -3500.586,E2 -3500.586} C_VEL
LIN {X 0,Y 545.897,Z 407.554,A -85,B 0,C 180,E1 -3500.786,E2 -3500.786} C_VEL
LIN {X 0,Y 545.675,Z 419.469,A -85,B 0,C 180,E1 -3501.389,E2 -3501.389} C_VEL
LIN {X 0,Y 545.455,Z 430.703,A -85,B 0,C 180,E1 -3502.132,E2 -3502.132} C_VEL
LIN {X 0,Y 545.258,Z 441.047,A -85,B 0,C 180,E1 -3502.971,E2 -3502.971} C_VEL
LIN {X 0,Y 545.129,Z 450.23,A -85,B 0,C 180,E1 -3503.895,E2 -3503.895} C_VEL
LIN {X 0,Y 544.952,Z 459.193,A -85,B 0,C 180,E1 -3505.006,E2 -3505.006} C_VEL
LIN {X 0,Y 544.837,Z 466.413,A -85,B 0,C 180,E1 -3506.117,E2 -3506.117} C_VEL
LIN {X 0,Y 544.724,Z 473.017,A -85,B 0,C 180,E1 -3507.412,E2 -3507.412} C_VEL
LIN {X 0,Y 544.642,Z 478.618,A -85,B 0,C 180,E1 -3508.891,E2 -3508.891} C_VEL
LIN {X 0,Y 544.547,Z 481.568,A -85,B 0,C 180,E1 -3510,E2 -3510} C_VEL
LIN {X 0,Y 544.543,Z 483.07,A -85,B 0,C 180,E1 -3510.74,E2 -3510.74} C_VEL
LIN {X 0,Y 544.57,Z 484.731,A -85,B 0,C 180,E1 -3512.219,E2 -3512.219} C_VEL
LIN {X 0,Y 544.645,Z 484.988,A -85,B 0,C 180,E1 -3512.959,E2 -3512.959} C_VEL
LIN {X 0,Y 544.646,Z 484.836,A -85,B 0,C 180,E1 -3513.699,E2 -3513.699} C_VEL
LIN {X 0,Y 544.603,Z 483.328,A -85,B 0,C 180,E1 -3515.183,E2 -3515.183} C_VEL
LIN {X 0,Y 544.654,Z 480.163,A -85,B 0,C 180,E1 -3516.669,E2 -3516.669} C_VEL
LIN {X 0,Y 544.672,Z 476.626,A -85,B 0,C 180,E1 -3517.787,E2 -3517.787} C_VEL
LIN {X 0,Y 544.712,Z 471.917,A -85,B 0,C 180,E1 -3518.907,E2 -3518.907} C_VEL
LIN {X 0,Y 544.832,Z 466,A -85,B 0,C 180,E1 -3520.029,E2 -3520.029} C_VEL
LIN {X 0,Y 544.909,Z 460.048,A -85,B 0,C 180,E1 -3520.967,E2 -3520.967} C_VEL
LIN {X 0,Y 545.031,Z 452.675,A -85,B 0,C 180,E1 -3521.907,E2 -3521.907} C_VEL
LIN {X 0,Y 545.164,Z 445.867,A -85,B 0,C 180,E1 -3522.66,E2 -3522.66} C_VEL
LIN {X 0,Y 545.317,Z 435.387,A -85,B 0,C 180,E1 -3523.604,E2 -3523.604} C_VEL
LIN {X 0,Y 545.583,Z 423.541,A -85,B 0,C 180,E1 -3524.453,E2 -3524.453} C_VEL
LIN {X 0,Y 545.829,Z 410.886,A -85,B 0,C 180,E1 -3525.153,E2 -3525.153} C_VEL
LIN {X 0,Y 545.698,Z 406.053,A -85,B 0,C 180,E1 -3525.376,E2 -3525.376} C_VEL
LIN {X 0,Y 545.143,Z 403.581,A -85,B 0,C 180,E1 -3525.497,E2 -3525.497} C_VEL
LIN {X 0,Y 545.08,Z 403.587,A -85,B 0,C 180,E1 -3528.805,E2 -3528.805} C_VEL
LIN {X 0,Y 545.07,Z 403.584,A -85,B 0,C 180,E1 -3531.163,E2 -3531.163} C_VEL
LIN {X 0,Y 545.055,Z 403.594,A -85,B 0,C 180,E1 -3534.369,E2 -3534.369} C_VEL
LIN {X 0,Y 545.086,Z 403.581,A -85,B 0,C 180,E1 -3537.171,E2 -3537.171} C_VEL
LIN {X 0,Y 545.07,Z 403.583,A -85,B 0,C 180,E1 -3539.338,E2 -3539.338} C_VEL
LIN {X 0,Y 545.06,Z 403.589,A -85,B 0,C 180,E1 -3541.915,E2 -3541.915} C_VEL
LIN {X 0,Y 545.084,Z 403.585,A -85,B 0,C 180,E1 -3544.563,E2 -3544.563} C_VEL
LIN {X 0,Y 545.043,Z 403.587,A -85,B 0,C 180,E1 -3547.304,E2 -3547.304} C_VEL
LIN {X 0,Y 545.071,Z 403.593,A -85,B 0,C 180,E1 -3550.143,E2 -3550.143} C_VEL
LIN {X 0,Y 545.083,Z 403.581,A -85,B 0,C 180,E1 -3553.107,E2 -3553.107} C_VEL
LIN {X 0,Y 545.065,Z 403.591,A -85,B 0,C 180,E1 -3556.225,E2 -3556.225} C_VEL
LIN {X 0,Y 545.093,Z 403.58,A -85,B 0,C 180,E1 -3558.886,E2 -3558.886} C_VEL
LIN {X 0,Y 545.057,Z 403.591,A -85,B 0,C 180,E1 -3561.763,E2 -3561.763} C_VEL
LIN {X 0,Y 545.041,Z 403.589,A -85,B 0,C 180,E1 -3564.532,E2 -3564.532} C_VEL
LIN {X 0,Y 545.074,Z 403.583,A -85,B 0,C 180,E1 -3567.212,E2 -3567.212} C_VEL
LIN {X 0,Y 545.069,Z 403.592,A -85,B 0,C 180,E1 -3569.81,E2 -3569.81} C_VEL
LIN {X 0,Y 545.083,Z 403.584,A -85,B 0,C 180,E1 -3572.344,E2 -3572.344} C_VEL
LIN {X 0,Y 545.122,Z 403.577,A -85,B 0,C 180,E1 -3574.82,E2 -3574.82} C_VEL
LIN {X 0,Y 545.041,Z 403.589,A -85,B 0,C 180,E1 -3577.242,E2 -3577.242} C_VEL
LIN {X 0,Y 545.122,Z 403.578,A -85,B 0,C 180,E1 -3580.415,E2 -3580.415} C_VEL
LIN {X 0,Y 545.069,Z 403.59,A -85,B 0,C 180,E1 -3583.521,E2 -3583.521} C_VEL
LIN {X 0,Y 545.099,Z 403.588,A -85,B 0,C 180,E1 -3585.82,E2 -3585.82} C_VEL
LIN {X 0,Y 545.152,Z 403.644,A -85,B 0,C 180,E1 -3588.602,E2 -3588.602} C_VEL
LIN {X 0,Y 545.852,Z 407.564,A -85,B 0,C 180,E1 -3588.79,E2 -3588.79} C_VEL
LIN {X 0,Y 545.769,Z 416.652,A -85,B 0,C 180,E1 -3589.238,E2 -3589.238} C_VEL
LIN {X 0,Y 545.577,Z 425.921,A -85,B 0,C 180,E1 -3589.798,E2 -3589.798} C_VEL
LIN {X 0,Y 545.355,Z 434.851,A -85,B 0,C 180,E1 -3590.449,E2 -3590.449} C_VEL
LIN {X 0,Y 545.255,Z 442.402,A -85,B 0,C 180,E1 -3591.102,E2 -3591.102} C_VEL
LIN {X 0,Y 545.101,Z 449.749,A -85,B 0,C 180,E1 -3591.846,E2 -3591.846} C_VEL
LIN {X 0,Y 544.95,Z 457.435,A -85,B 0,C 180,E1 -3592.776,E2 -3592.776} C_VEL
LIN {X 0,Y 544.868,Z 462.898,A -85,B 0,C 180,E1 -3593.552,E2 -3593.552} C_VEL
LIN {X 0,Y 544.766,Z 468.239,A -85,B 0,C 180,E1 -3594.447,E2 -3594.447} C_VEL
LIN {X 0,Y 544.718,Z 473.624,A -85,B 0,C 180,E1 -3595.56,E2 -3595.56} C_VEL
LIN {X 0,Y 544.708,Z 477.852,A -85,B 0,C 180,E1 -3596.671,E2 -3596.671} C_VEL
LIN {X 0,Y 544.588,Z 481.034,A -85,B 0,C 180,E1 -3597.781,E2 -3597.781} C_VEL
LIN {X 0,Y 544.551,Z 482.661,A -85,B 0,C 180,E1 -3598.521,E2 -3598.521} C_VEL
LIN {X 0,Y 544.543,Z 483.83,A -85,B 0,C 180,E1 -3599.26,E2 -3599.26} C_VEL
LIN {X 0,Y 544.541,Z 484.932,A -85,B 0,C 180,E1 -3600.739,E2 -3600.739} C_VEL
LIN {X 0,Y 544.545,Z 484.919,A -85,B 0,C 180,E1 -3601.479,E2 -3601.479} C_VEL
LIN {X 0,Y 544.646,Z 483.632,A -85,B 0,C 180,E1 -3602.959,E2 -3602.959} C_VEL
LIN {X 0,Y 544.653,Z 482.432,A -85,B 0,C 180,E1 -3603.699,E2 -3603.699} C_VEL
LIN {X 0,Y 544.601,Z 479.787,A -85,B 0,C 180,E1 -3604.812,E2 -3604.812} C_VEL
LIN {X 0,Y 544.706,Z 476.126,A -85,B 0,C 180,E1 -3605.924,E2 -3605.924} C_VEL
LIN {X 0,Y 544.735,Z 471.336,A -85,B 0,C 180,E1 -3607.04,E2 -3607.04} C_VEL
LIN {X 0,Y 544.827,Z 465.256,A -85,B 0,C 180,E1 -3608.157,E2 -3608.157} C_VEL
LIN {X 0,Y 544.92,Z 459.083,A -85,B 0,C 180,E1 -3609.09,E2 -3609.09} C_VEL
LIN {X 0,Y 545.02,Z 453.292,A -85,B 0,C 180,E1 -3609.838,E2 -3609.838} C_VEL
LIN {X 0,Y 545.197,Z 446.546,A -85,B 0,C 180,E1 -3610.585,E2 -3610.585} C_VEL
LIN {X 0,Y 545.264,Z 437.212,A -85,B 0,C 180,E1 -3611.448,E2 -3611.448} C_VEL
LIN {X 0,Y 545.508,Z 428.94,A -85,B 0,C 180,E1 -3612.085,E2 -3612.085} C_VEL
LIN {X 0,Y 545.647,Z 420.242,A -85,B 0,C 180,E1 -3612.648,E2 -3612.648} C_VEL
LIN {X 0,Y 545.809,Z 410.492,A -85,B 0,C 180,E1 -3613.165,E2 -3613.165} C_VEL
LIN {X 0,Y 545.735,Z 406.416,A -85,B 0,C 180,E1 -3613.356,E2 -3613.356} C_VEL
LIN {X 0,Y 545.084,Z 403.59,A -85,B 0,C 180,E1 -3613.515,E2 -3613.515} C_VEL
LIN {X 0,Y 545.065,Z 403.591,A -85,B 0,C 180,E1 -3615.71,E2 -3615.71} C_VEL
LIN {X 0,Y 545.075,Z 403.591,A -85,B 0,C 180,E1 -3618.026,E2 -3618.026} C_VEL
LIN {X 0,Y 545.1,Z 403.59,A -85,B 0,C 180,E1 -3620.372,E2 -3620.372} C_VEL
LIN {X 0,Y 545.083,Z 403.588,A -85,B 0,C 180,E1 -3623.559,E2 -3623.559} C_VEL
LIN {X 0,Y 545.085,Z 403.589,A -85,B 0,C 180,E1 -3626,E2 -3626} C_VEL
LIN {X 0,Y 545.094,Z 403.588,A -85,B 0,C 180,E1 -3628.748,E2 -3628.748} C_VEL
LIN {X 0,Y 545.062,Z 403.591,A -85,B 0,C 180,E1 -3631.679,E2 -3631.679} C_VEL
LIN {X 0,Y 545.066,Z 403.59,A -85,B 0,C 180,E1 -3634.564,E2 -3634.564} C_VEL
LIN {X 0,Y 545.04,Z 403.593,A -85,B 0,C 180,E1 -3637.304,E2 -3637.304} C_VEL
LIN {X 0,Y 545.07,Z 403.59,A -85,B 0,C 180,E1 -3640.142,E2 -3640.142} C_VEL
LIN {X 0,Y 545.091,Z 403.586,A -85,B 0,C 180,E1 -3643.106,E2 -3643.106} C_VEL
LIN {X 0,Y 545.053,Z 403.591,A -85,B 0,C 180,E1 -3646.226,E2 -3646.226} C_VEL
LIN {X 0,Y 545.095,Z 403.587,A -85,B 0,C 180,E1 -3648.886,E2 -3648.886} C_VEL
LIN {X 0,Y 545.058,Z 403.593,A -85,B 0,C 180,E1 -3651.763,E2 -3651.763} C_VEL
LIN {X 0,Y 545.107,Z 403.716,A -85,B 0,C 180,E1 -3652.498,E2 -3652.498} C_VEL
LIN {X 0,Y 546.319,Z 410.682,A -85,B 0,C 180,E1 -3654.14,E2 -3654.14} C_VEL
LIN {X 0,Y 546.09,Z 421.129,A -85,B 0,C 180,E1 -3656.399,E2 -3656.399} C_VEL
LIN {X 0,Y 546.001,Z 435.326,A -85,B 0,C 180,E1 -3659.341,E2 -3659.341} C_VEL
LIN {X 0,Y 545.89,Z 449.547,A -85,B 0,C 180,E1 -3662.18,E2 -3662.18} C_VEL
LIN {X 0,Y 545.761,Z 464.31,A -85,B 0,C 180,E1 -3665.056,E2 -3665.056} C_VEL
LIN {X 0,Y 545.652,Z 477.956,A -85,B 0,C 180,E1 -3667.669,E2 -3667.669} C_VEL
LIN {X 0,Y 545.527,Z 492.712,A -85,B 0,C 180,E1 -3670.43,E2 -3670.43} C_VEL
LIN {X 0,Y 545.28,Z 506.447,A -85,B 0,C 180,E1 -3673.142,E2 -3673.142} C_VEL
LIN {X 0,Y 545.067,Z 522.098,A -85,B 0,C 180,E1 -3676.2,E2 -3676.2} C_VEL
LIN {X 0,Y 545.013,Z 525.155,A -85,B 0,C 180,E1 -3676.792,E2 -3676.792} C_VEL
LIN {X 0,Y 546.184,Z 533.217,A -85,B 0,C 180,E1 -3676.963,E2 -3676.963} C_VEL
LIN {X 0,Y 546.039,Z 546.494,A -85,B 0,C 180,E1 -3677.314,E2 -3677.314} C_VEL
LIN {X 0,Y 545.879,Z 558.508,A -85,B 0,C 180,E1 -3677.782,E2 -3677.782} C_VEL
LIN {X 0,Y 545.708,Z 570.367,A -85,B 0,C 180,E1 -3678.401,E2 -3678.401} C_VEL
LIN {X 0,Y 545.455,Z 581.482,A -85,B 0,C 180,E1 -3679.138,E2 -3679.138} C_VEL
LIN {X 0,Y 545.276,Z 591.644,A -85,B 0,C 180,E1 -3679.979,E2 -3679.979} C_VEL
LIN {X 0,Y 545.082,Z 600.784,A -85,B 0,C 180,E1 -3680.912,E2 -3680.912} C_VEL
LIN {X 0,Y 544.917,Z 609.687,A -85,B 0,C 180,E1 -3682.03,E2 -3682.03} C_VEL
LIN {X 0,Y 544.785,Z 616.848,A -85,B 0,C 180,E1 -3683.146,E2 -3683.146} C_VEL
LIN {X 0,Y 544.741,Z 623.365,A -85,B 0,C 180,E1 -3684.447,E2 -3684.447} C_VEL
LIN {X 0,Y 544.66,Z 627.676,A -85,B 0,C 180,E1 -3685.559,E2 -3685.559} C_VEL
LIN {X 0,Y 544.669,Z 629.958,A -85,B 0,C 180,E1 -3686.301,E2 -3686.301} C_VEL
LIN {X 0,Y 544.65,Z 631.807,A -85,B 0,C 180,E1 -3687.041,E2 -3687.041} C_VEL
LIN {X 0,Y 544.546,Z 634.184,A -85,B 0,C 180,E1 -3688.521,E2 -3688.521} C_VEL
LIN {X 0,Y 544.541,Z 635,A -85,B 0,C 180,E1 -3690,E2 -3690} C_VEL
LIN {X 0,Y 544.546,Z 634.185,A -85,B 0,C 180,E1 -3691.479,E2 -3691.479} C_VEL
LIN {X 0,Y 544.65,Z 631.81,A -85,B 0,C 180,E1 -3692.958,E2 -3692.958} C_VEL
LIN {X 0,Y 544.683,Z 628.896,A -85,B 0,C 180,E1 -3694.069,E2 -3694.069} C_VEL
LIN {X 0,Y 544.654,Z 624.949,A -85,B 0,C 180,E1 -3695.182,E2 -3695.182} C_VEL
LIN {X 0,Y 544.739,Z 619.704,A -85,B 0,C 180,E1 -3696.328,E2 -3696.328} C_VEL
LIN {X 0,Y 544.836,Z 613.468,A -85,B 0,C 180,E1 -3697.411,E2 -3697.411} C_VEL
LIN {X 0,Y 545.006,Z 605.479,A -85,B 0,C 180,E1 -3698.528,E2 -3698.528} C_VEL
LIN {X 0,Y 545.142,Z 597.335,A -85,B 0,C 180,E1 -3699.461,E2 -3699.461} C_VEL
LIN {X 0,Y 545.364,Z 587.4,A -85,B 0,C 180,E1 -3700.394,E2 -3700.394} C_VEL
LIN {X 0,Y 545.566,Z 576.596,A -85,B 0,C 180,E1 -3701.208,E2 -3701.208} C_VEL
LIN {X 0,Y 545.746,Z 565.176,A -85,B 0,C 180,E1 -3701.891,E2 -3701.891} C_VEL
LIN {X 0,Y 545.933,Z 552.978,A -85,B 0,C 180,E1 -3702.452,E2 -3702.452} C_VEL
LIN {X 0,Y 546.108,Z 540.179,A -85,B 0,C 180,E1 -3702.873,E2 -3702.873} C_VEL
LIN {X 0,Y 546.003,Z 531.378,A -85,B 0,C 180,E1 -3703.08,E2 -3703.08} C_VEL
LIN {X 0,Y 545.023,Z 525.035,A -85,B 0,C 180,E1 -3703.231,E2 -3703.231} C_VEL
LIN {X 0,Y 545.229,Z 510.362,A -85,B 0,C 180,E1 -3706.089,E2 -3706.089} C_VEL
LIN {X 0,Y 545.429,Z 496.667,A -85,B 0,C 180,E1 -3708.792,E2 -3708.792} C_VEL
LIN {X 0,Y 545.569,Z 484.305,A -85,B 0,C 180,E1 -3711.143,E2 -3711.143} C_VEL
LIN {X 0,Y 545.728,Z 469.829,A -85,B 0,C 180,E1 -3713.886,E2 -3713.886} C_VEL
LIN {X 0,Y 545.853,Z 455.903,A -85,B 0,C 180,E1 -3716.578,E2 -3716.578} C_VEL
LIN {X 0,Y 545.993,Z 440.144,A -85,B 0,C 180,E1 -3719.707,E2 -3719.707} C_VEL
LIN {X 0,Y 546.079,Z 425.39,A -85,B 0,C 180,E1 -3722.72,E2 -3722.72} C_VEL
LIN {X 0,Y 546.342,Z 411.705,A -85,B 0,C 180,E1 -3725.617,E2 -3725.617} C_VEL
LIN {X 0,Y 545.511,Z 405.703,A -85,B 0,C 180,E1 -3726.987,E2 -3726.987} C_VEL
LIN {X 0,Y 545.062,Z 403.593,A -85,B 0,C 180,E1 -3727.534,E2 -3727.534} C_VEL
LIN {X 0,Y 545.112,Z 403.587,A -85,B 0,C 180,E1 -3730.476,E2 -3730.476} C_VEL
LIN {X 0,Y 545.08,Z 403.59,A -85,B 0,C 180,E1 -3733.106,E2 -3733.106} C_VEL
LIN {X 0,Y 545.067,Z 403.591,A -85,B 0,C 180,E1 -3736.224,E2 -3736.224} C_VEL
LIN {X 0,Y 545.1,Z 403.588,A -85,B 0,C 180,E1 -3738.887,E2 -3738.887} C_VEL
LIN {X 0,Y 545.056,Z 403.592,A -85,B 0,C 180,E1 -3741.763,E2 -3741.763} C_VEL
LIN {X 0,Y 545.054,Z 403.594,A -85,B 0,C 180,E1 -3744.533,E2 -3744.533} C_VEL
LIN {X 0,Y 545.07,Z 403.589,A -85,B 0,C 180,E1 -3747.212,E2 -3747.212} C_VEL
LIN {X 0,Y 545.066,Z 403.592,A -85,B 0,C 180,E1 -3749.811,E2 -3749.811} C_VEL
LIN {X 0,Y 545.099,Z 403.587,A -85,B 0,C 180,E1 -3752.345,E2 -3752.345} C_VEL
LIN {X 0,Y 545.121,Z 403.584,A -85,B 0,C 180,E1 -3754.821,E2 -3754.821} C_VEL
LIN {X 0,Y 545.047,Z 403.594,A -85,B 0,C 180,E1 -3757.243,E2 -3757.243} C_VEL
LIN {X 0,Y 545.123,Z 403.585,A -85,B 0,C 180,E1 -3760.415,E2 -3760.415} C_VEL
LIN {X 0,Y 545.077,Z 403.589,A -85,B 0,C 180,E1 -3763.521,E2 -3763.521} C_VEL
LIN {X 0,Y 545.098,Z 403.587,A -85,B 0,C 180,E1 -3765.82,E2 -3765.82} C_VEL
LIN {X 0,Y 545.12,Z 403.583,A -85,B 0,C 180,E1 -3768.849,E2 -3768.849} C_VEL
LIN {X 0,Y 545.1,Z 403.587,A -85,B 0,C 180,E1 -3771.847,E2 -3771.847} C_VEL
LIN {X 0,Y 545.209,Z 403.574,A -85,B 0,C 180,E1 -3774.823,E2 -3774.823} C_VEL
LIN {X 0,Y 545.201,Z 403.575,A -85,B 0,C 180,E1 -3777.784,E2 -3777.784} C_VEL
LIN {X 0,Y 545.218,Z 403.571,A -85,B 0,C 180,E1 -3780.739,E2 -3780.739} C_VEL
LIN {X 0,Y 545.175,Z 403.576,A -85,B 0,C 180,E1 -3782.956,E2 -3782.956} C_VEL
LIN {X 0,Y 545.172,Z 403.579,A -85,B 0,C 180,E1 -3785.92,E2 -3785.92} C_VEL
LIN {X 0,Y 545.125,Z 403.585,A -85,B 0,C 180,E1 -3788.9,E2 -3788.9} C_VEL
LIN {X 0,Y 545.138,Z 403.583,A -85,B 0,C 180,E1 -3791.904,E2 -3791.904} C_VEL
LIN {X 0,Y 545.088,Z 403.587,A -85,B 0,C 180,E1 -3794.944,E2 -3794.944} C_VEL
LIN {X 0,Y 545.082,Z 403.589,A -85,B 0,C 180,E1 -3798.026,E2 -3798.026} C_VEL
LIN {X 0,Y 545.102,Z 403.587,A -85,B 0,C 180,E1 -3800.372,E2 -3800.372} C_VEL
LIN {X 0,Y 545.095,Z 403.587,A -85,B 0,C 180,E1 -3803.559,E2 -3803.559} C_VEL
LIN {X 0,Y 545.082,Z 403.59,A -85,B 0,C 180,E1 -3806.001,E2 -3806.001} C_VEL
LIN {X 0,Y 545.092,Z 403.587,A -85,B 0,C 180,E1 -3808.748,E2 -3808.748} C_VEL
LIN {X 0,Y 545.062,Z 403.594,A -85,B 0,C 180,E1 -3811.679,E2 -3811.679} C_VEL
LIN {X 0,Y 545.081,Z 403.589,A -85,B 0,C 180,E1 -3814.563,E2 -3814.563} C_VEL
LIN {X 0,Y 545.068,Z 403.591,A -85,B 0,C 180,E1 -3817.012,E2 -3817.012} C_VEL
LIN {X 0,Y 544.36,Z 403.68,A -85,B 0,C 180,E1 -3817.629,E2 -3817.629} C_VEL
LIN {X 0,Y 541.492,Z 404.036,A -85,B 0,C 180,E1 -3818.629,E2 -3818.629} C_VEL
LIN {X 0,Y 539.104,Z 404.335,A -85,B 0,C 180,E1 -3819.435,E2 -3819.435} C_VEL
LIN {X 0,Y 538.095,Z 404.46,A -85,B 0,C 180,E1 -3820.057,E2 -3820.057} C_VEL
LIN {X 0,Y 538.02,Z 404.466,A -85,B 0,C 180,E1 -3820.268,E2 -3820.268} C_VEL
LIN {X 0,Y 538.037,Z 404.465,A -85,B 0,C 180,E1 -3822.989,E2 -3822.989} C_VEL
LIN {X 0,Y 538.033,Z 404.468,A -85,B 0,C 180,E1 -3825.926,E2 -3825.926} C_VEL
LIN {X 0,Y 538.055,Z 404.465,A -85,B 0,C 180,E1 -3829.225,E2 -3829.225} C_VEL
LIN {X 0,Y 537.997,Z 404.474,A -85,B 0,C 180,E1 -3832.123,E2 -3832.123} C_VEL
LIN {X 0,Y 538.02,Z 404.467,A -85,B 0,C 180,E1 -3834.917,E2 -3834.917} C_VEL
LIN {X 0,Y 538.036,Z 404.469,A -85,B 0,C 180,E1 -3837.619,E2 -3837.619} C_VEL
LIN {X 0,Y 538.048,Z 404.465,A -85,B 0,C 180,E1 -3840.241,E2 -3840.241} C_VEL
LIN {X 0,Y 538.067,Z 404.463,A -85,B 0,C 180,E1 -3842.796,E2 -3842.796} C_VEL
LIN {X 0,Y 538.053,Z 404.467,A -85,B 0,C 180,E1 -3845.293,E2 -3845.293} C_VEL
LIN {X 0,Y 538.027,Z 404.468,A -85,B 0,C 180,E1 -3848.546,E2 -3848.546} C_VEL
LIN {X 0,Y 538.044,Z 404.466,A -85,B 0,C 180,E1 -3850.94,E2 -3850.94} C_VEL
LIN {X 0,Y 538.028,Z 404.468,A -85,B 0,C 180,E1 -3853.299,E2 -3853.299} C_VEL
LIN {X 0,Y 538.069,Z 404.463,A -85,B 0,C 180,E1 -3855.631,E2 -3855.631} C_VEL
LIN {X 0,Y 538.083,Z 404.461,A -85,B 0,C 180,E1 -3858.702,E2 -3858.702} C_VEL
LIN {X 0,Y 538.064,Z 404.511,A -85,B 0,C 180,E1 -3860.461,E2 -3860.461} C_VEL
LIN {X 0,Y 538.936,Z 408.524,A -85,B 0,C 180,E1 -3860.666,E2 -3860.666} C_VEL
LIN {X 0,Y 538.705,Z 420.149,A -85,B 0,C 180,E1 -3861.277,E2 -3861.277} C_VEL
LIN {X 0,Y 538.452,Z 431.254,A -85,B 0,C 180,E1 -3862.029,E2 -3862.029} C_VEL
LIN {X 0,Y 538.233,Z 441.972,A -85,B 0,C 180,E1 -3862.923,E2 -3862.923} C_VEL
LIN {X 0,Y 538.085,Z 450.569,A -85,B 0,C 180,E1 -3863.814,E2 -3863.814} C_VEL
LIN {X 0,Y 537.903,Z 459.486,A -85,B 0,C 180,E1 -3864.941,E2 -3864.941} C_VEL
LIN {X 0,Y 537.757,Z 466.634,A -85,B 0,C 180,E1 -3866.066,E2 -3866.066} C_VEL
LIN {X 0,Y 537.632,Z 473.201,A -85,B 0,C 180,E1 -3867.378,E2 -3867.378} C_VEL
LIN {X 0,Y 537.559,Z 478.741,A -85,B 0,C 180,E1 -3868.876,E2 -3868.876} C_VEL
LIN {X 0,Y 537.448,Z 481.642,A -85,B 0,C 180,E1 -3870,E2 -3870} C_VEL
LIN {X 0,Y 537.443,Z 483.138,A -85,B 0,C 180,E1 -3870.749,E2 -3870.749} C_VEL
LIN {X 0,Y 537.489,Z 484.755,A -85,B 0,C 180,E1 -3872.248,E2 -3872.248} C_VEL
LIN {X 0,Y 537.545,Z 484.996,A -85,B 0,C 180,E1 -3872.998,E2 -3872.998} C_VEL
LIN {X 0,Y 537.562,Z 484.811,A -85,B 0,C 180,E1 -3873.748,E2 -3873.748} C_VEL
LIN {X 0,Y 537.524,Z 483.27,A -85,B 0,C 180,E1 -3875.251,E2 -3875.251} C_VEL
LIN {X 0,Y 537.557,Z 480.053,A -85,B 0,C 180,E1 -3876.758,E2 -3876.758} C_VEL
LIN {X 0,Y 537.579,Z 476.479,A -85,B 0,C 180,E1 -3877.89,E2 -3877.89} C_VEL
LIN {X 0,Y 537.637,Z 471.716,A -85,B 0,C 180,E1 -3879.025,E2 -3879.025} C_VEL
LIN {X 0,Y 537.753,Z 465.753,A -85,B 0,C 180,E1 -3880.162,E2 -3880.162} C_VEL
LIN {X 0,Y 537.873,Z 459.758,A -85,B 0,C 180,E1 -3881.112,E2 -3881.112} C_VEL
LIN {X 0,Y 538.024,Z 450.745,A -85,B 0,C 180,E1 -3882.255,E2 -3882.255} C_VEL
LIN {X 0,Y 538.214,Z 441.522,A -85,B 0,C 180,E1 -3883.21,E2 -3883.21} C_VEL
LIN {X 0,Y 538.457,Z 431.138,A -85,B 0,C 180,E1 -3884.07,E2 -3884.07} C_VEL
LIN {X 0,Y 538.659,Z 421.504,A -85,B 0,C 180,E1 -3884.722,E2 -3884.722} C_VEL
LIN {X 0,Y 538.891,Z 411.281,A -85,B 0,C 180,E1 -3885.294,E2 -3885.294} C_VEL
LIN {X 0,Y 538.826,Z 407.598,A -85,B 0,C 180,E1 -3885.47,E2 -3885.47} C_VEL
LIN {X 0,Y 538.078,Z 404.462,A -85,B 0,C 180,E1 -3885.652,E2 -3885.652} C_VEL
LIN {X 0,Y 538.031,Z 404.469,A -85,B 0,C 180,E1 -3888.27,E2 -3888.27} C_VEL
LIN {X 0,Y 538.043,Z 404.465,A -85,B 0,C 180,E1 -3890.651,E2 -3890.651} C_VEL
LIN {X 0,Y 538.008,Z 404.466,A -85,B 0,C 180,E1 -3893.888,E2 -3893.888} C_VEL
LIN {X 0,Y 538.045,Z 404.467,A -85,B 0,C 180,E1 -3896.367,E2 -3896.367} C_VEL
LIN {X 0,Y 538.036,Z 404.461,A -85,B 0,C 180,E1 -3898.933,E2 -3898.933} C_VEL
LIN {X 0,Y 538.015,Z 404.466,A -85,B 0,C 180,E1 -3901.887,E2 -3901.887} C_VEL
LIN {X 0,Y 538.033,Z 404.463,A -85,B 0,C 180,E1 -3904.62,E2 -3904.62} C_VEL
LIN {X 0,Y 538.011,Z 404.462,A -85,B 0,C 180,E1 -3907.17,E2 -3907.17} C_VEL
LIN {X 0,Y 538.028,Z 404.465,A -85,B 0,C 180,E1 -3909.797,E2 -3909.797} C_VEL
LIN {X 0,Y 538.023,Z 404.462,A -85,B 0,C 180,E1 -3912.786,E2 -3912.786} C_VEL
LIN {X 0,Y 538.032,Z 404.467,A -85,B 0,C 180,E1 -3915.926,E2 -3915.926} C_VEL
LIN {X 0,Y 538.054,Z 404.458,A -85,B 0,C 180,E1 -3919.224,E2 -3919.224} C_VEL
LIN {X 0,Y 537.997,Z 404.472,A -85,B 0,C 180,E1 -3922.122,E2 -3922.122} C_VEL
LIN {X 0,Y 538.003,Z 404.464,A -85,B 0,C 180,E1 -3924.916,E2 -3924.916} C_VEL
LIN {X 0,Y 538.024,Z 404.466,A -85,B 0,C 180,E1 -3927.617,E2 -3927.617} C_VEL
LIN {X 0,Y 538.022,Z 404.465,A -85,B 0,C 180,E1 -3930.239,E2 -3930.239} C_VEL
LIN {X 0,Y 538.058,Z 404.457,A -85,B 0,C 180,E1 -3932.796,E2 -3932.796} C_VEL
LIN {X 0,Y 538.032,Z 404.462,A -85,B 0,C 180,E1 -3935.292,E2 -3935.292} C_VEL
LIN {X 0,Y 538.02,Z 404.467,A -85,B 0,C 180,E1 -3938.042,E2 -3938.042} C_VEL
LIN {X 0,Y 538.037,Z 404.46,A -85,B 0,C 180,E1 -3940.94,E2 -3940.94} C_VEL
LIN {X 0,Y 538.017,Z 404.465,A -85,B 0,C 180,E1 -3943.299,E2 -3943.299} C_VEL
LIN {X 0,Y 538.069,Z 404.464,A -85,B 0,C 180,E1 -3945.631,E2 -3945.631} C_VEL
LIN {X 0,Y 538.102,Z 404.538,A -85,B 0,C 180,E1 -3948.467,E2 -3948.467} C_VEL
LIN {X 0,Y 538.846,Z 407.976,A -85,B 0,C 180,E1 -3948.647,E2 -3948.647} C_VEL
LIN {X 0,Y 538.804,Z 416.877,A -85,B 0,C 180,E1 -3949.098,E2 -3949.098} C_VEL
LIN {X 0,Y 538.596,Z 426.106,A -85,B 0,C 180,E1 -3949.664,E2 -3949.664} C_VEL
LIN {X 0,Y 538.36,Z 435.007,A -85,B 0,C 180,E1 -3950.324,E2 -3950.324} C_VEL
LIN {X 0,Y 538.235,Z 442.534,A -85,B 0,C 180,E1 -3950.985,E2 -3950.985} C_VEL
LIN {X 0,Y 538.06,Z 449.861,A -85,B 0,C 180,E1 -3951.739,E2 -3951.739} C_VEL
LIN {X 0,Y 537.898,Z 457.527,A -85,B 0,C 180,E1 -3952.681,E2 -3952.681} C_VEL
LIN {X 0,Y 537.805,Z 463.441,A -85,B 0,C 180,E1 -3953.544,E2 -3953.544} C_VEL
LIN {X 0,Y 537.712,Z 468.301,A -85,B 0,C 180,E1 -3954.374,E2 -3954.374} C_VEL
LIN {X 0,Y 537.624,Z 473.674,A -85,B 0,C 180,E1 -3955.501,E2 -3955.501} C_VEL
LIN {X 0,Y 537.636,Z 477.89,A -85,B 0,C 180,E1 -3956.628,E2 -3956.628} C_VEL
LIN {X 0,Y 537.505,Z 481.061,A -85,B 0,C 180,E1 -3957.752,E2 -3957.752} C_VEL
LIN {X 0,Y 537.456,Z 482.675,A -85,B 0,C 180,E1 -3958.501,E2 -3958.501} C_VEL
LIN {X 0,Y 537.443,Z 483.849,A -85,B 0,C 180,E1 -3959.251,E2 -3959.251} C_VEL
LIN {X 0,Y 537.441,Z 484.925,A -85,B 0,C 180,E1 -3960.749,E2 -3960.749} C_VEL
LIN {X 0,Y 537.451,Z 484.917,A -85,B 0,C 180,E1 -3961.499,E2 -3961.499} C_VEL
LIN {X 0,Y 537.547,Z 483.603,A -85,B 0,C 180,E1 -3962.998,E2 -3962.998} C_VEL
LIN {X 0,Y 537.57,Z 482.408,A -85,B 0,C 180,E1 -3963.748,E2 -3963.748} C_VEL
LIN {X 0,Y 537.517,Z 479.751,A -85,B 0,C 180,E1 -3964.875,E2 -3964.875} C_VEL
LIN {X 0,Y 537.615,Z 476.075,A -85,B 0,C 180,E1 -3966.003,E2 -3966.003} C_VEL
LIN {X 0,Y 537.655,Z 471.257,A -85,B 0,C 180,E1 -3967.133,E2 -3967.133} C_VEL
LIN {X 0,Y 537.753,Z 465.161,A -85,B 0,C 180,E1 -3968.265,E2 -3968.265} C_VEL
LIN {X 0,Y 537.881,Z 458.974,A -85,B 0,C 180,E1 -3969.21,E2 -3969.21} C_VEL
LIN {X 0,Y 537.991,Z 453.164,A -85,B 0,C 180,E1 -3969.967,E2 -3969.967} C_VEL
LIN {X 0,Y 538.178,Z 446.395,A -85,B 0,C 180,E1 -3970.725,E2 -3970.725} C_VEL
LIN {X 0,Y 538.252,Z 437.844,A -85,B 0,C 180,E1 -3971.531,E2 -3971.531} C_VEL
LIN {X 0,Y 538.513,Z 428.724,A -85,B 0,C 180,E1 -3972.244,E2 -3972.244} C_VEL
LIN {X 0,Y 538.704,Z 419.983,A -85,B 0,C 180,E1 -3972.814,E2 -3972.814} C_VEL
LIN {X 0,Y 538.89,Z 409.206,A -85,B 0,C 180,E1 -3973.385,E2 -3973.385} C_VEL
LIN {X 0,Y 538.045,Z 404.466,A -85,B 0,C 180,E1 -3973.647,E2 -3973.647} C_VEL
LIN {X 0,Y 538.03,Z 404.47,A -85,B 0,C 180,E1 -3975.921,E2 -3975.921} C_VEL
LIN {X 0,Y 538.03,Z 404.468,A -85,B 0,C 180,E1 -3978.27,E2 -3978.27} C_VEL
LIN {X 0,Y 538.044,Z 404.467,A -85,B 0,C 180,E1 -3980.651,E2 -3980.651} C_VEL
LIN {X 0,Y 538.006,Z 404.47,A -85,B 0,C 180,E1 -3983.888,E2 -3983.888} C_VEL
LIN {X 0,Y 538.047,Z 404.464,A -85,B 0,C 180,E1 -3986.366,E2 -3986.366} C_VEL
LIN {X 0,Y 538.035,Z 404.466,A -85,B 0,C 180,E1 -3988.933,E2 -3988.933} C_VEL
LIN {X 0,Y 538.014,Z 404.468,A -85,B 0,C 180,E1 -3991.887,E2 -3991.887} C_VEL
LIN {X 0,Y 538.016,Z 404.468,A -85,B 0,C 180,E1 -3994.617,E2 -3994.617} C_VEL
LIN {X 0,Y 538.008,Z 404.47,A -85,B 0,C 180,E1 -3997.17,E2 -3997.17} C_VEL
LIN {X 0,Y 538.027,Z 404.47,A -85,B 0,C 180,E1 -3999.797,E2 -3999.797} C_VEL
LIN {X 0,Y 538.037,Z 404.466,A -85,B 0,C 180,E1 -4002.988,E2 -4002.988} C_VEL
LIN {X 0,Y 538.023,Z 404.466,A -85,B 0,C 180,E1 -4005.926,E2 -4005.926} C_VEL
LIN {X 0,Y 538.054,Z 404.465,A -85,B 0,C 180,E1 -4009.224,E2 -4009.224} C_VEL
LIN {X 0,Y 538.05,Z 404.597,A -85,B 0,C 180,E1 -4012.258,E2 -4012.258} C_VEL
LIN {X 0,Y 539.416,Z 412.277,A -85,B 0,C 180,E1 -4014.105,E2 -4014.105} C_VEL
LIN {X 0,Y 539.179,Z 424.638,A -85,B 0,C 180,E1 -4016.807,E2 -4016.807} C_VEL
LIN {X 0,Y 538.974,Z 440.322,A -85,B 0,C 180,E1 -4020.081,E2 -4020.081} C_VEL
LIN {X 0,Y 538.827,Z 455.075,A -85,B 0,C 180,E1 -4023.047,E2 -4023.047} C_VEL
LIN {X 0,Y 538.688,Z 469.903,A -85,B 0,C 180,E1 -4025.96,E2 -4025.96} C_VEL
LIN {X 0,Y 538.507,Z 485.482,A -85,B 0,C 180,E1 -4028.967,E2 -4028.967} C_VEL
LIN {X 0,Y 538.351,Z 500.235,A -85,B 0,C 180,E1 -4031.741,E2 -4031.741} C_VEL
LIN {X 0,Y 538.19,Z 512.316,A -85,B 0,C 180,E1 -4034.084,E2 -4034.084} C_VEL
LIN {X 0,Y 537.976,Z 525.155,A -85,B 0,C 180,E1 -4036.616,E2 -4036.616} C_VEL
LIN {X 0,Y 539.301,Z 534.357,A -85,B 0,C 180,E1 -4036.817,E2 -4036.817} C_VEL
LIN {X 0,Y 539.127,Z 546.495,A -85,B 0,C 180,E1 -4037.148,E2 -4037.148} C_VEL
LIN {X 0,Y 538.925,Z 558.506,A -85,B 0,C 180,E1 -4037.622,E2 -4037.622} C_VEL
LIN {X 0,Y 538.757,Z 570.145,A -85,B 0,C 180,E1 -4038.236,E2 -4038.236} C_VEL
LIN {X 0,Y 538.463,Z 581.483,A -85,B 0,C 180,E1 -4038.995,E2 -4038.995} C_VEL
LIN {X 0,Y 538.272,Z 591.644,A -85,B 0,C 180,E1 -4039.848,E2 -4039.848} C_VEL
LIN {X 0,Y 538.055,Z 600.784,A -85,B 0,C 180,E1 -4040.792,E2 -4040.792} C_VEL
LIN {X 0,Y 537.851,Z 609.687,A -85,B 0,C 180,E1 -4041.925,E2 -4041.925} C_VEL
LIN {X 0,Y 537.729,Z 616.847,A -85,B 0,C 180,E1 -4043.056,E2 -4043.056} C_VEL
LIN {X 0,Y 537.676,Z 623.365,A -85,B 0,C 180,E1 -4044.374,E2 -4044.374} C_VEL
LIN {X 0,Y 537.558,Z 627.676,A -85,B 0,C 180,E1 -4045.501,E2 -4045.501} C_VEL
LIN {X 0,Y 537.591,Z 629.958,A -85,B 0,C 180,E1 -4046.252,E2 -4046.252} C_VEL
LIN {X 0,Y 537.551,Z 631.807,A -85,B 0,C 180,E1 -4047.002,E2 -4047.002} C_VEL
LIN {X 0,Y 537.451,Z 634.183,A -85,B 0,C 180,E1 -4048.501,E2 -4048.501} C_VEL
LIN {X 0,Y 537.442,Z 635,A -85,B 0,C 180,E1 -4050,E2 -4050} C_VEL
LIN {X 0,Y 537.451,Z 634.185,A -85,B 0,C 180,E1 -4051.498,E2 -4051.498} C_VEL
LIN {X 0,Y 537.551,Z 631.81,A -85,B 0,C 180,E1 -4052.998,E2 -4052.998} C_VEL
LIN {X 0,Y 537.603,Z 628.896,A -85,B 0,C 180,E1 -4054.123,E2 -4054.123} C_VEL
LIN {X 0,Y 537.588,Z 624.949,A -85,B 0,C 180,E1 -4055.25,E2 -4055.25} C_VEL
LIN {X 0,Y 537.65,Z 620.08,A -85,B 0,C 180,E1 -4056.335,E2 -4056.335} C_VEL
LIN {X 0,Y 537.79,Z 613.468,A -85,B 0,C 180,E1 -4057.509,E2 -4057.509} C_VEL
LIN {X 0,Y 537.972,Z 605.478,A -85,B 0,C 180,E1 -4058.64,E2 -4058.64} C_VEL
LIN {X 0,Y 538.118,Z 597.335,A -85,B 0,C 180,E1 -4059.585,E2 -4059.585} C_VEL
LIN {X 0,Y 538.361,Z 587.399,A -85,B 0,C 180,E1 -4060.531,E2 -4060.531} C_VEL
LIN {X 0,Y 538.574,Z 577.592,A -85,B 0,C 180,E1 -4061.288,E2 -4061.288} C_VEL
LIN {X 0,Y 538.754,Z 566.548,A -85,B 0,C 180,E1 -4061.973,E2 -4061.973} C_VEL
LIN {X 0,Y 538.982,Z 554.106,A -85,B 0,C 180,E1 -4062.568,E2 -4062.568} C_VEL
LIN {X 0,Y 539.184,Z 541.091,A -85,B 0,C 180,E1 -4063.018,E2 -4063.018} C_VEL
LIN {X 0,Y 539.158,Z 532.659,A -85,B 0,C 180,E1 -4063.222,E2 -4063.222} C_VEL
LIN {X 0,Y 537.971,Z 525.035,A -85,B 0,C 180,E1 -4063.408,E2 -4063.408} C_VEL
LIN {X 0,Y 538.214,Z 510.362,A -85,B 0,C 180,E1 -4066.305,E2 -4066.305} C_VEL
LIN {X 0,Y 538.375,Z 498.151,A -85,B 0,C 180,E1 -4068.652,E2 -4068.652} C_VEL
LIN {X 0,Y 538.526,Z 483.397,A -85,B 0,C 180,E1 -4071.433,E2 -4071.433} C_VEL
LIN {X 0,Y 538.694,Z 468.517,A -85,B 0,C 180,E1 -4074.317,E2 -4074.317} C_VEL
LIN {X 0,Y 538.831,Z 455.142,A -85,B 0,C 180,E1 -4076.952,E2 -4076.952} C_VEL
LIN {X 0,Y 538.993,Z 440.431,A -85,B 0,C 180,E1 -4079.917,E2 -4079.917} C_VEL
LIN {X 0,Y 539.109,Z 426.742,A -85,B 0,C 180,E1 -4082.752,E2 -4082.752} C_VEL
LIN {X 0,Y 539.405,Z 413.162,A -85,B 0,C 180,E1 -4085.666,E2 -4085.666} C_VEL
LIN {X 0,Y 538.73,Z 407.909,A -85,B 0,C 180,E1 -4086.877,E2 -4086.877} C_VEL
LIN {X 0,Y 538.027,Z 404.469,A -85,B 0,C 180,E1 -4087.741,E2 -4087.741} C_VEL
LIN {X 0,Y 538.079,Z 404.462,A -85,B 0,C 180,E1 -4090.773,E2 -4090.773} C_VEL
LIN {X 0,Y 538.021,Z 404.47,A -85,B 0,C 180,E1 -4094.073,E2 -4094.073} C_VEL
LIN {X 0,Y 538.035,Z 404.469,A -85,B 0,C 180,E1 -4097.012,E2 -4097.012} C_VEL
LIN {X 0,Y 538.054,Z 404.465,A -85,B 0,C 180,E1 -4099.252,E2 -4099.252} C_VEL
LIN {X 0,Y 537.996,Z 404.473,A -85,B 0,C 180,E1 -4102.122,E2 -4102.122} C_VEL
LIN {X 0,Y 538.014,Z 404.469,A -85,B 0,C 180,E1 -4104.917,E2 -4104.917} C_VEL
LIN {X 0,Y 538.02,Z 404.469,A -85,B 0,C 180,E1 -4107.617,E2 -4107.617} C_VEL
LIN {X 0,Y 538.019,Z 404.469,A -85,B 0,C 180,E1 -4110.239,E2 -4110.239} C_VEL
LIN {X 0,Y 538.074,Z 404.462,A -85,B 0,C 180,E1 -4112.797,E2 -4112.797} C_VEL
LIN {X 0,Y 538.052,Z 404.465,A -85,B 0,C 180,E1 -4115.293,E2 -4115.293} C_VEL
LIN {X 0,Y 538.017,Z 404.469,A -85,B 0,C 180,E1 -4118.042,E2 -4118.042} C_VEL
LIN {X 0,Y 538.04,Z 404.466,A -85,B 0,C 180,E1 -4120.94,E2 -4120.94} C_VEL
LIN {X 0,Y 538.028,Z 404.467,A -85,B 0,C 180,E1 -4123.299,E2 -4123.299} C_VEL
LIN {X 0,Y 538.067,Z 404.462,A -85,B 0,C 180,E1 -4125.631,E2 -4125.631} C_VEL
LIN {X 0,Y 538.08,Z 404.461,A -85,B 0,C 180,E1 -4128.702,E2 -4128.702} C_VEL
LIN {X 0,Y 538.064,Z 404.465,A -85,B 0,C 180,E1 -4131.739,E2 -4131.739} C_VEL
LIN {X 0,Y 538.127,Z 404.456,A -85,B 0,C 180,E1 -4134.003,E2 -4134.003} C_VEL
LIN {X 0,Y 538.145,Z 404.454,A -85,B 0,C 180,E1 -4137.006,E2 -4137.006} C_VEL
LIN {X 0,Y 538.174,Z 404.45,A -85,B 0,C 180,E1 -4140,E2 -4140} C_VEL
LIN {X 0,Y 538.141,Z 404.452,A -85,B 0,C 180,E1 -4142.995,E2 -4142.995} C_VEL
LIN {X 0,Y 538.125,Z 404.456,A -85,B 0,C 180,E1 -4145.997,E2 -4145.997} C_VEL
LIN {X 0,Y 538.075,Z 404.462,A -85,B 0,C 180,E1 -4149.018,E2 -4149.018} C_VEL
LIN {X 0,Y 538.087,Z 404.463,A -85,B 0,C 180,E1 -4152.063,E2 -4152.063} C_VEL
LIN {X 0,Y 538.048,Z 404.465,A -85,B 0,C 180,E1 -4155.144,E2 -4155.144} C_VEL
LIN {X 0,Y 538.034,Z 404.467,A -85,B 0,C 180,E1 -4158.27,E2 -4158.27} C_VEL
LIN {X 0,Y 538.046,Z 404.467,A -85,B 0,C 180,E1 -4160.651,E2 -4160.651} C_VEL
LIN {X 0,Y 538.027,Z 404.469,A -85,B 0,C 180,E1 -4163.888,E2 -4163.888} C_VEL
LIN {X 0,Y 538.045,Z 404.466,A -85,B 0,C 180,E1 -4166.367,E2 -4166.367} C_VEL
LIN {X 0,Y 538.033,Z 404.465,A -85,B 0,C 180,E1 -4168.934,E2 -4168.934} C_VEL
LIN {X 0,Y 538.017,Z 404.47,A -85,B 0,C 180,E1 -4171.888,E2 -4171.888} C_VEL
LIN {X 0,Y 538.031,Z 404.468,A -85,B 0,C 180,E1 -4174.62,E2 -4174.62} C_VEL
LIN {X 0,Y 538.011,Z 404.471,A -85,B 0,C 180,E1 -4177.171,E2 -4177.171} C_VEL
LIN {X 0,Y 538.02,Z 404.466,A -85,B 0,C 180,E1 -4180.268,E2 -4180.268} C_VEL
LIN {X 0,Y 537.373,Z 404.548,A -85,B 0,C 180,E1 -4180.893,E2 -4180.893} C_VEL
LIN {X 0,Y 534.525,Z 404.906,A -85,B 0,C 180,E1 -4181.908,E2 -4181.908} C_VEL
LIN {X 0,Y 532.103,Z 405.21,A -85,B 0,C 180,E1 -4182.725,E2 -4182.725} C_VEL
LIN {X 0,Y 531.055,Z 405.338,A -85,B 0,C 180,E1 -4183.356,E2 -4183.356} C_VEL
LIN {X 0,Y 530.967,Z 405.348,A -85,B 0,C 180,E1 -4183.57,E2 -4183.57} C_VEL
LIN {X 0,Y 530.97,Z 405.347,A -85,B 0,C 180,E1 -4186.506,E2 -4186.506} C_VEL
LIN {X 0,Y 530.993,Z 405.345,A -85,B 0,C 180,E1 -4188.976,E2 -4188.976} C_VEL
LIN {X 0,Y 530.962,Z 405.348,A -85,B 0,C 180,E1 -4191.53,E2 -4191.53} C_VEL
LIN {X 0,Y 530.983,Z 405.346,A -85,B 0,C 180,E1 -4194.382,E2 -4194.382} C_VEL
LIN {X 0,Y 530.977,Z 405.345,A -85,B 0,C 180,E1 -4197.134,E2 -4197.134} C_VEL
LIN {X 0,Y 530.991,Z 405.346,A -85,B 0,C 180,E1 -4199.804,E2 -4199.804} C_VEL
LIN {X 0,Y 531.019,Z 405.34,A -85,B 0,C 180,E1 -4202.467,E2 -4202.467} C_VEL
LIN {X 0,Y 531.01,Z 405.341,A -85,B 0,C 180,E1 -4204.943,E2 -4204.943} C_VEL
LIN {X 0,Y 530.976,Z 405.347,A -85,B 0,C 180,E1 -4208.247,E2 -4208.247} C_VEL
LIN {X 0,Y 531.002,Z 405.343,A -85,B 0,C 180,E1 -4210.678,E2 -4210.678} C_VEL
LIN {X 0,Y 530.99,Z 405.345,A -85,B 0,C 180,E1 -4213.071,E2 -4213.071} C_VEL
LIN {X 0,Y 531.024,Z 405.34,A -85,B 0,C 180,E1 -4215.436,E2 -4215.436} C_VEL
LIN {X 0,Y 531.043,Z 405.338,A -85,B 0,C 180,E1 -4218.55,E2 -4218.55} C_VEL
LIN {X 0,Y 531.03,Z 405.412,A -85,B 0,C 180,E1 -4220.285,E2 -4220.285} C_VEL
LIN {X 0,Y 532.05,Z 409.398,A -85,B 0,C 180,E1 -4220.496,E2 -4220.496} C_VEL
LIN {X 0,Y 531.835,Z 421.753,A -85,B 0,C 180,E1 -4221.163,E2 -4221.163} C_VEL
LIN {X 0,Y 531.508,Z 433.898,A -85,B 0,C 180,E1 -4222.019,E2 -4222.019} C_VEL
LIN {X 0,Y 531.206,Z 445.299,A -85,B 0,C 180,E1 -4223.057,E2 -4223.057} C_VEL
LIN {X 0,Y 530.994,Z 452.944,A -85,B 0,C 180,E1 -4223.922,E2 -4223.922} C_VEL
LIN {X 0,Y 530.869,Z 460.084,A -85,B 0,C 180,E1 -4224.873,E2 -4224.873} C_VEL
LIN {X 0,Y 530.698,Z 467.008,A -85,B 0,C 180,E1 -4226.013,E2 -4226.013} C_VEL
LIN {X 0,Y 530.546,Z 473.382,A -85,B 0,C 180,E1 -4227.343,E2 -4227.343} C_VEL
LIN {X 0,Y 530.478,Z 478.864,A -85,B 0,C 180,E1 -4228.861,E2 -4228.861} C_VEL
LIN {X 0,Y 530.349,Z 481.716,A -85,B 0,C 180,E1 -4230,E2 -4230} C_VEL
LIN {X 0,Y 530.345,Z 483.202,A -85,B 0,C 180,E1 -4230.759,E2 -4230.759} C_VEL
LIN {X 0,Y 530.41,Z 484.779,A -85,B 0,C 180,E1 -4232.278,E2 -4232.278} C_VEL
LIN {X 0,Y 530.45,Z 485,A -85,B 0,C 180,E1 -4233.038,E2 -4233.038} C_VEL
LIN {X 0,Y 530.48,Z 484.786,A -85,B 0,C 180,E1 -4233.798,E2 -4233.798} C_VEL
LIN {X 0,Y 530.447,Z 483.211,A -85,B 0,C 180,E1 -4235.322,E2 -4235.322} C_VEL
LIN {X 0,Y 530.476,Z 479.943,A -85,B 0,C 180,E1 -4236.848,E2 -4236.848} C_VEL
LIN {X 0,Y 530.508,Z 476.333,A -85,B 0,C 180,E1 -4237.996,E2 -4237.996} C_VEL
LIN {X 0,Y 530.547,Z 471.56,A -85,B 0,C 180,E1 -4239.147,E2 -4239.147} C_VEL
LIN {X 0,Y 530.708,Z 465.705,A -85,B 0,C 180,E1 -4240.299,E2 -4240.299} C_VEL
LIN {X 0,Y 530.839,Z 459.789,A -85,B 0,C 180,E1 -4241.261,E2 -4241.261} C_VEL
LIN {X 0,Y 531.047,Z 450.929,A -85,B 0,C 180,E1 -4242.419,E2 -4242.419} C_VEL
LIN {X 0,Y 531.255,Z 441.757,A -85,B 0,C 180,E1 -4243.386,E2 -4243.386} C_VEL
LIN {X 0,Y 531.561,Z 431.447,A -85,B 0,C 180,E1 -4244.256,E2 -4244.256} C_VEL
LIN {X 0,Y 531.796,Z 422.455,A -85,B 0,C 180,E1 -4244.878,E2 -4244.878} C_VEL
LIN {X 0,Y 532.029,Z 411.472,A -85,B 0,C 180,E1 -4245.496,E2 -4245.496} C_VEL
LIN {X 0,Y 531.635,Z 407.741,A -85,B 0,C 180,E1 -4245.685,E2 -4245.685} C_VEL
LIN {X 0,Y 531.006,Z 405.345,A -85,B 0,C 180,E1 -4245.812,E2 -4245.812} C_VEL
LIN {X 0,Y 530.991,Z 405.346,A -85,B 0,C 180,E1 -4248.521,E2 -4248.521} C_VEL
LIN {X 0,Y 531.004,Z 405.338,A -85,B 0,C 180,E1 -4250.938,E2 -4250.938} C_VEL
LIN {X 0,Y 530.971,Z 405.347,A -85,B 0,C 180,E1 -4254.225,E2 -4254.225} C_VEL
LIN {X 0,Y 531.003,Z 405.338,A -85,B 0,C 180,E1 -4256.744,E2 -4256.744} C_VEL
LIN {X 0,Y 530.987,Z 405.338,A -85,B 0,C 180,E1 -4259.323,E2 -4259.323} C_VEL
LIN {X 0,Y 530.971,Z 405.347,A -85,B 0,C 180,E1 -4262.1,E2 -4262.1} C_VEL
LIN {X 0,Y 530.989,Z 405.338,A -85,B 0,C 180,E1 -4264.853,E2 -4264.853} C_VEL
LIN {X 0,Y 530.971,Z 405.341,A -85,B 0,C 180,E1 -4267.508,E2 -4267.508} C_VEL
LIN {X 0,Y 530.986,Z 405.342,A -85,B 0,C 180,E1 -4270.433,E2 -4270.433} C_VEL
LIN {X 0,Y 530.966,Z 405.34,A -85,B 0,C 180,E1 -4273.281,E2 -4273.281} C_VEL
LIN {X 0,Y 530.992,Z 405.34,A -85,B 0,C 180,E1 -4275.621,E2 -4275.621} C_VEL
LIN {X 0,Y 531.003,Z 405.338,A -85,B 0,C 180,E1 -4278.565,E2 -4278.565} C_VEL
LIN {X 0,Y 530.962,Z 405.344,A -85,B 0,C 180,E1 -4281.529,E2 -4281.529} C_VEL
LIN {X 0,Y 530.959,Z 405.344,A -85,B 0,C 180,E1 -4284.38,E2 -4284.38} C_VEL
LIN {X 0,Y 530.972,Z 405.34,A -85,B 0,C 180,E1 -4287.133,E2 -4287.133} C_VEL
LIN {X 0,Y 530.975,Z 405.347,A -85,B 0,C 180,E1 -4289.803,E2 -4289.803} C_VEL
LIN {X 0,Y 531.016,Z 405.335,A -85,B 0,C 180,E1 -4292.468,E2 -4292.468} C_VEL
LIN {X 0,Y 530.999,Z 405.336,A -85,B 0,C 180,E1 -4294.942,E2 -4294.942} C_VEL
LIN {X 0,Y 530.976,Z 405.342,A -85,B 0,C 180,E1 -4298.247,E2 -4298.247} C_VEL
LIN {X 0,Y 530.997,Z 405.336,A -85,B 0,C 180,E1 -4300.677,E2 -4300.677} C_VEL
LIN {X 0,Y 530.975,Z 405.34,A -85,B 0,C 180,E1 -4303.07,E2 -4303.07} C_VEL
LIN {X 0,Y 531.024,Z 405.338,A -85,B 0,C 180,E1 -4305.436,E2 -4305.436} C_VEL
LIN {X 0,Y 531.084,Z 405.5,A -85,B 0,C 180,E1 -4308.314,E2 -4308.314} C_VEL
LIN {X 0,Y 531.985,Z 410.409,A -85,B 0,C 180,E1 -4308.57,E2 -4308.57} C_VEL
LIN {X 0,Y 531.857,Z 421.009,A -85,B 0,C 180,E1 -4309.146,E2 -4309.146} C_VEL
LIN {X 0,Y 531.544,Z 430.93,A -85,B 0,C 180,E1 -4309.814,E2 -4309.814} C_VEL
LIN {X 0,Y 531.264,Z 441.228,A -85,B 0,C 180,E1 -4310.674,E2 -4310.674} C_VEL
LIN {X 0,Y 531.061,Z 450.37,A -85,B 0,C 180,E1 -4311.629,E2 -4311.629} C_VEL
LIN {X 0,Y 530.878,Z 457.903,A -85,B 0,C 180,E1 -4312.584,E2 -4312.584} C_VEL
LIN {X 0,Y 530.741,Z 464.152,A -85,B 0,C 180,E1 -4313.535,E2 -4313.535} C_VEL
LIN {X 0,Y 530.663,Z 468.446,A -85,B 0,C 180,E1 -4314.299,E2 -4314.299} C_VEL
LIN {X 0,Y 530.529,Z 473.723,A -85,B 0,C 180,E1 -4315.441,E2 -4315.441} C_VEL
LIN {X 0,Y 530.536,Z 477.928,A -85,B 0,C 180,E1 -4316.582,E2 -4316.582} C_VEL
LIN {X 0,Y 530.427,Z 481.089,A -85,B 0,C 180,E1 -4317.722,E2 -4317.722} C_VEL
LIN {X 0,Y 530.366,Z 482.69,A -85,B 0,C 180,E1 -4318.481,E2 -4318.481} C_VEL
LIN {X 0,Y 530.345,Z 483.867,A -85,B 0,C 180,E1 -4319.241,E2 -4319.241} C_VEL
LIN {X 0,Y 530.343,Z 484.918,A -85,B 0,C 180,E1 -4320.759,E2 -4320.759} C_VEL
LIN {X 0,Y 530.361,Z 484.914,A -85,B 0,C 180,E1 -4321.519,E2 -4321.519} C_VEL
LIN {X 0,Y 530.452,Z 483.575,A -85,B 0,C 180,E1 -4323.038,E2 -4323.038} C_VEL
LIN {X 0,Y 530.488,Z 482.384,A -85,B 0,C 180,E1 -4323.798,E2 -4323.798} C_VEL
LIN {X 0,Y 530.438,Z 479.714,A -85,B 0,C 180,E1 -4324.94,E2 -4324.94} C_VEL
LIN {X 0,Y 530.504,Z 476.019,A -85,B 0,C 180,E1 -4326.084,E2 -4326.084} C_VEL
LIN {X 0,Y 530.577,Z 471.231,A -85,B 0,C 180,E1 -4327.229,E2 -4327.229} C_VEL
LIN {X 0,Y 530.7,Z 465.275,A -85,B 0,C 180,E1 -4328.376,E2 -4328.376} C_VEL
LIN {X 0,Y 530.864,Z 459.208,A -85,B 0,C 180,E1 -4329.333,E2 -4329.333} C_VEL
LIN {X 0,Y 530.993,Z 453.495,A -85,B 0,C 180,E1 -4330.1,E2 -4330.1} C_VEL
LIN {X 0,Y 531.218,Z 446.81,A -85,B 0,C 180,E1 -4330.867,E2 -4330.867} C_VEL
LIN {X 0,Y 531.356,Z 437.562,A -85,B 0,C 180,E1 -4331.752,E2 -4331.752} C_VEL
LIN {X 0,Y 531.642,Z 427.974,A -85,B 0,C 180,E1 -4332.502,E2 -4332.502} C_VEL
LIN {X 0,Y 531.903,Z 417.344,A -85,B 0,C 180,E1 -4333.175,E2 -4333.175} C_VEL
LIN {X 0,Y 531.831,Z 408.801,A -85,B 0,C 180,E1 -4333.614,E2 -4333.614} C_VEL
LIN {X 0,Y 531.042,Z 405.337,A -85,B 0,C 180,E1 -4333.806,E2 -4333.806} C_VEL
LIN {X 0,Y 530.98,Z 405.345,A -85,B 0,C 180,E1 -4336.929,E2 -4336.929} C_VEL
LIN {X 0,Y 531.029,Z 405.343,A -85,B 0,C 180,E1 -4340.127,E2 -4340.127} C_VEL
LIN {X 0,Y 530.949,Z 405.35,A -85,B 0,C 180,E1 -4342.573,E2 -4342.573} C_VEL
LIN {X 0,Y 530.999,Z 405.342,A -85,B 0,C 180,E1 -4345.058,E2 -4345.058} C_VEL
LIN {X 0,Y 531.02,Z 405.339,A -85,B 0,C 180,E1 -4347.595,E2 -4347.595} C_VEL
LIN {X 0,Y 530.978,Z 405.344,A -85,B 0,C 180,E1 -4350.645,E2 -4350.645} C_VEL
LIN {X 0,Y 530.991,Z 405.343,A -85,B 0,C 180,E1 -4353.773,E2 -4353.773} C_VEL
LIN {X 0,Y 530.959,Z 405.348,A -85,B 0,C 180,E1 -4356.558,E2 -4356.558} C_VEL
LIN {X 0,Y 530.989,Z 405.344,A -85,B 0,C 180,E1 -4359.443,E2 -4359.443} C_VEL
LIN {X 0,Y 530.984,Z 405.346,A -85,B 0,C 180,E1 -4362.456,E2 -4362.456} C_VEL
LIN {X 0,Y 530.986,Z 405.343,A -85,B 0,C 180,E1 -4365.621,E2 -4365.621} C_VEL
LIN {X 0,Y 531,Z 405.343,A -85,B 0,C 180,E1 -4368.565,E2 -4368.565} C_VEL
LIN {X 0,Y 530.963,Z 405.349,A -85,B 0,C 180,E1 -4371.529,E2 -4371.529} C_VEL
LIN {X 0,Y 530.991,Z 405.466,A -85,B 0,C 180,E1 -4372.015,E2 -4372.015} C_VEL
LIN {X 0,Y 532.313,Z 412.072,A -85,B 0,C 180,E1 -4373.646,E2 -4373.646} C_VEL
LIN {X 0,Y 532.46,Z 417.603,A -85,B 0,C 180,E1 -4374.92,E2 -4374.92} C_VEL
LIN {X 0,Y 532.09,Z 432.285,A -85,B 0,C 180,E1 -4378.107,E2 -4378.107} C_VEL
LIN {X 0,Y 531.938,Z 445.867,A -85,B 0,C 180,E1 -4380.952,E2 -4380.952} C_VEL
LIN {X 0,Y 531.774,Z 459.368,A -85,B 0,C 180,E1 -4383.686,E2 -4383.686} C_VEL
LIN {X 0,Y 531.582,Z 474.22,A -85,B 0,C 180,E1 -4386.632,E2 -4386.632} C_VEL
LIN {X 0,Y 531.397,Z 488.834,A -85,B 0,C 180,E1 -4389.483,E2 -4389.483} C_VEL
LIN {X 0,Y 531.261,Z 504.546,A -85,B 0,C 180,E1 -4392.485,E2 -4392.485} C_VEL
LIN {X 0,Y 531.035,Z 520.099,A -85,B 0,C 180,E1 -4395.436,E2 -4395.436} C_VEL
LIN {X 0,Y 530.932,Z 525.155,A -85,B 0,C 180,E1 -4396.435,E2 -4396.435} C_VEL
LIN {X 0,Y 532.4,Z 535.497,A -85,B 0,C 180,E1 -4396.668,E2 -4396.668} C_VEL
LIN {X 0,Y 532.174,Z 547.867,A -85,B 0,C 180,E1 -4397.026,E2 -4397.026} C_VEL
LIN {X 0,Y 531.97,Z 559.498,A -85,B 0,C 180,E1 -4397.506,E2 -4397.506} C_VEL
LIN {X 0,Y 531.77,Z 571.091,A -85,B 0,C 180,E1 -4398.137,E2 -4398.137} C_VEL
LIN {X 0,Y 531.483,Z 581.482,A -85,B 0,C 180,E1 -4398.849,E2 -4398.849} C_VEL
LIN {X 0,Y 531.23,Z 591.644,A -85,B 0,C 180,E1 -4399.712,E2 -4399.712} C_VEL
LIN {X 0,Y 531.012,Z 600.784,A -85,B 0,C 180,E1 -4400.669,E2 -4400.669} C_VEL
LIN {X 0,Y 530.813,Z 609.686,A -85,B 0,C 180,E1 -4401.817,E2 -4401.817} C_VEL
LIN {X 0,Y 530.664,Z 616.847,A -85,B 0,C 180,E1 -4402.963,E2 -4402.963} C_VEL
LIN {X 0,Y 530.611,Z 623.365,A -85,B 0,C 180,E1 -4404.299,E2 -4404.299} C_VEL
LIN {X 0,Y 530.457,Z 627.676,A -85,B 0,C 180,E1 -4405.44,E2 -4405.44} C_VEL
LIN {X 0,Y 530.516,Z 629.958,A -85,B 0,C 180,E1 -4406.202,E2 -4406.202} C_VEL
LIN {X 0,Y 530.457,Z 631.807,A -85,B 0,C 180,E1 -4406.962,E2 -4406.962} C_VEL
LIN {X 0,Y 530.41,Z 633.194,A -85,B 0,C 180,E1 -4407.722,E2 -4407.722} C_VEL
LIN {X 0,Y 530.344,Z 634.786,A -85,B 0,C 180,E1 -4409.241,E2 -4409.241} C_VEL
LIN {X 0,Y 530.342,Z 635,A -85,B 0,C 180,E1 -4410,E2 -4410} C_VEL
LIN {X 0,Y 530.361,Z 634.184,A -85,B 0,C 180,E1 -4411.519,E2 -4411.519} C_VEL
LIN {X 0,Y 530.41,Z 633.197,A -85,B 0,C 180,E1 -4412.278,E2 -4412.278} C_VEL
LIN {X 0,Y 530.457,Z 631.81,A -85,B 0,C 180,E1 -4413.038,E2 -4413.038} C_VEL
LIN {X 0,Y 530.522,Z 628.896,A -85,B 0,C 180,E1 -4414.178,E2 -4414.178} C_VEL
LIN {X 0,Y 530.525,Z 624.949,A -85,B 0,C 180,E1 -4415.321,E2 -4415.321} C_VEL
LIN {X 0,Y 530.599,Z 619.263,A -85,B 0,C 180,E1 -4416.582,E2 -4416.582} C_VEL
LIN {X 0,Y 530.758,Z 612.236,A -85,B 0,C 180,E1 -4417.8,E2 -4417.8} C_VEL
LIN {X 0,Y 530.931,Z 603.993,A -85,B 0,C 180,E1 -4418.948,E2 -4418.948} C_VEL
LIN {X 0,Y 531.113,Z 595.541,A -85,B 0,C 180,E1 -4419.905,E2 -4419.905} C_VEL
LIN {X 0,Y 531.402,Z 585.093,A -85,B 0,C 180,E1 -4420.863,E2 -4420.863} C_VEL
LIN {X 0,Y 531.692,Z 574.36,A -85,B 0,C 180,E1 -4421.656,E2 -4421.656} C_VEL
LIN {X 0,Y 531.933,Z 563.406,A -85,B 0,C 180,E1 -4422.301,E2 -4422.301} C_VEL
LIN {X 0,Y 532.091,Z 551.767,A -85,B 0,C 180,E1 -4422.83,E2 -4422.83} C_VEL
LIN {X 0,Y 532.33,Z 538.348,A -85,B 0,C 180,E1 -4423.261,E2 -4423.261} C_VEL
LIN {X 0,Y 532.13,Z 532.789,A -85,B 0,C 180,E1 -4423.397,E2 -4423.397} C_VEL
LIN {X 0,Y 530.944,Z 525.035,A -85,B 0,C 180,E1 -4423.589,E2 -4423.589} C_VEL
LIN {X 0,Y 531.152,Z 510.822,A -85,B 0,C 180,E1 -4426.33,E2 -4426.33} C_VEL
LIN {X 0,Y 531.309,Z 496.203,A -85,B 0,C 180,E1 -4429.11,E2 -4429.11} C_VEL
LIN {X 0,Y 531.506,Z 481.204,A -85,B 0,C 180,E1 -4431.989,E2 -4431.989} C_VEL
LIN {X 0,Y 531.676,Z 466.933,A -85,B 0,C 180,E1 -4434.815,E2 -4434.815} C_VEL
LIN {X 0,Y 531.865,Z 452.529,A -85,B 0,C 180,E1 -4437.708,E2 -4437.708} C_VEL
LIN {X 0,Y 532.02,Z 439.006,A -85,B 0,C 180,E1 -4440.485,E2 -4440.485} C_VEL
LIN {X 0,Y 532.162,Z 425.981,A -85,B 0,C 180,E1 -4443.235,E2 -4443.235} C_VEL
